TYPE UDT 31
VERSION : 0.0
  STRUCT
   A_FD_OR : BYTE ;	//Feedrate override
   A_DriveEnable : BOOL ;	//Drive test movement enable
   A_AckFixedStop : BOOL ;	//Acknowledge fixed stop reached
   A_SensorFixedStop : BOOL ;	//Sensor fixed stop
   A_ASpDisable : BOOL ;	//Axis/spindle disable
   A_Follow_upMode : BOOL ;	//Follow-up mode
   A_PosMeas1 : BOOL ;	//Position measuring system 1
   A_PosMeas2 : BOOL ;	//Position measuring system 2
   A_ORactive : BOOL ;	//Override active
   A_SWCam : BOOL ;	//SW cam activation
   A_ContrEnable : BOOL ;	//Controller enable
   A_DelDTGSpReset : BOOL ;	//Delete distance to go/Spindle-Reset
   A_Clamp : BOOL ;	//Clamping in progress
   A_RefVal1 : BOOL ;	//Reference point value 1
   A_RefVal2 : BOOL ;	//Reference point value 2
   A_RefVal3 : BOOL ;	//Reference point value 3
   A_RefVal4 : BOOL ;	//Reference point value 4
   A_ExtZO : BOOL ;	//Import external ZO
   A_EnabTravFixedStop : BOOL ;	//Enable travel to fixed stop
   A_FixedFD1 : BOOL ;	//Activate fixed feed 1
   A_FixedFD2 : BOOL ;	//Activate fixed feed 2
   A_FixedFD3 : BOOL ;	//Activate fixed feed 3
   A_FixedFD4 : BOOL ;	//Activate fixed feed 4
   A_VelocSpeedLimit : BOOL ;	//Velocity/spindle speed limitation
   A_PrgtestAxRel : BOOL ;	// Program test axis/spindle release
   A_HW1 : BOOL ;	//Activate handwheel 1
   A_HW2 : BOOL ;	//Activate handwheel 2
   A_HW3 : BOOL ;	//Activate handwheel 3
   A_FDSpStop : BOOL ;	//Feed stop/spindle stop
   A_Disable : BOOL ;	//Traversing key disable
   A_RapidTrOR : BOOL ;	//Rapid traverse override
   A_Minus : BOOL ;	//Traversing key minus
   A_Plus : BOOL ;	//Traversing key plus
   A_INC1 : BOOL ;	//INC1
   A_INC10 : BOOL ;	//INC10
   A_INC100 : BOOL ;	//INC100
   A_INC1000 : BOOL ;	//INC1000
   A_INC10000 : BOOL ;	//INC10000
   A_INCVar : BOOL ;	//INC variable
   A_OEMAxis : BYTE ;	//OEM axis signals
   A_InvHWDirOfRot : BOOL ;	// Inverting handwheel direction of rotation
   f7_1 : BOOL ;
   f7_2 : BOOL ;
   f7_3 : BOOL ;
   f7_4 : BOOL ;
   f7_5 : BOOL ;
   f7_6 : BOOL ;
   f7_7 : BOOL ;
   A_NCASpChanA : BOOL ;	//Assign NC axis/spindle channel A
   A_NCASpChanB : BOOL ;	//Assign NC axis/spindle channel B
   A_NCASpChanC : BOOL ;	//Assign NC axis/spindle channel C
   A_NCASpChanD : BOOL ;	//Assign NC axis/spindle channel D
   A_NCASpStrobe : BOOL ;	//Activation of assignment with pos. edge
   f8_5 : BOOL ;
   f8_6 : BOOL ;
   A_PLCASp : BOOL ;	//Request PLC axis/spindle
   A_Para_A : BOOL ;	//Parameter block servo A
   A_Para_B : BOOL ;	//Parameter block servo B
   A_Para_C : BOOL ;	//Parameter block servo C
   A_LockParSetDef : BOOL ;	//Lock parameter set definition from NC
   f9_4 : BOOL ;
   f9_5 : BOOL ;
   f9_6 : BOOL ;
   f9_7 : BOOL ;
   A_REPOSDelay : BOOL ;	//REPOS DELAY
   f10_1 : BOOL ;
   f10_2 : BOOL ;
   f10_3 : BOOL ;
   f10_4 : BOOL ;
   f10_5 : BOOL ;
   f10_6 : BOOL ;
   f10_7 : BOOL ;
   A_StartBrakeTest : BOOL ;	// Start brake test
   f11_1 : BOOL ;
   f11_2 : BOOL ;
   f11_3 : BOOL ;
   f11_4 : BOOL ;
   f11_5 : BOOL ;
   f11_6 : BOOL ;
   f11_7 : BOOL ;
   A_HWLimitMinus : BOOL ;	//Hardware limit switch minus
   A_HWLimitPlus : BOOL ;	//Hardware limit switch plus
   A_SWLimit2Minus : BOOL ;	//2nd software limit switch minus
   A_SWLimit2Plus : BOOL ;	//2nd software limit switch plus
   A_ModuloLimitEn : BOOL ;	// Modulo limit enabled
   f12_5 : BOOL ;
   f12_6 : BOOL ;
   A_DelayRef : BOOL ;	//Delay reference point approach
   A_JogFixPPos0 : BOOL ;	// JogFixPointPos 0
   A_JogFixPPos1 : BOOL ;	// JogFixPointPos 1
   A_JogFixPPos2 : BOOL ;	// JogFixPointPos 2
   A_JogToPos : BOOL ;	// Jog to position
   f13_4 : BOOL ;
   f13_5 : BOOL ;
   f13_6 : BOOL ;
   f13_7 : BOOL ;
   A_ProgtestSuppress : BOOL ;	// Program test to supress
   A_ProgtestActivate : BOOL ;	// Program test activate
   f14_2 : BOOL ;
   f14_3 : BOOL ;
   f14_4 : BOOL ;
   f14_5 : BOOL ;
   f14_6 : BOOL ;
   f14_7 : BOOL ;
   f15 : BYTE ;
   A_ActGearA : BOOL ;	//Actual gear stage A
   A_ActGearB : BOOL ;	//Actual gear stage B
   A_ActGearC : BOOL ;	//Actual gear stage C
   A_GearChangeOv : BOOL ;	//Gear has changed over
   A_Sp1Syn : BOOL ;	//Re-synchronize spindle 1
   A_Sp2Syn : BOOL ;	//Re-synchronize spindle 2
   A_NoMonitorGear : BOOL ;	//No monitoring when changing gear
   A_DeleteS : BOOL ;	//Delete S value
   A_FD_ORSp : BOOL ;	//Feedrate override for spindle valid
   f17_1 : BOOL ;
   f17_2 : BOOL ;
   f17_3 : BOOL ;
   A_Sp1SynP : BOOL ;	//Re-synchronize spindle 1 f. positioning
   A_Sp2SynP : BOOL ;	//Re-synchronize spindle 2 f. positioning
   A_M3M4Inv : BOOL ;	//Invert M3/M4
   f17_7 : BOOL ;
   f18_0 : BOOL ;
   f18_1 : BOOL ;
   f18_2 : BOOL ;
   f18_3 : BOOL ;
   A_OscilPLC : BOOL ;	//Oscillation via PLC
   A_OscilSpeed : BOOL ;	//enable Oscillation
   A_SetRotDirectRight : BOOL ;	//Setpoint osci. direct. right
   A_SetRotDirectLeft : BOOL ;	//Setpoint osci. direct. left
   A_SpOR : BYTE ;	//Spindle override
   f20_0 : BOOL ;
   A_RUEncQuStop : BOOL ;	//Run-up encoder quick stop
   f20_2 : BOOL ;
   A_SpeedSetpSmooth : BOOL ;	//Speed setpoint smoothing
   f20_4 : BOOL ;
   A_HoldBrakeToOpen : BOOL ;	// holding brake open
   f20_6 : BOOL ;
   f20_7 : BOOL ;
   A_ParA : BOOL ;	//Parameter set selection A
   A_ParB : BOOL ;	//Parameter set selection B
   A_ParC : BOOL ;	//Parameter set selection C
   A_MotA : BOOL ;	//Motor selection A
   A_MotB : BOOL ;	//Motor selection B
   A_MotOK : BOOL ;	//Motor selected
   A_IntegratDisable : BOOL ;	//n controller integrator disable
   A_PulseEnable : BOOL ;	//Pulse enable
   A_SG_SBH : BOOL ;	//Deselection SG/SBH
   A_SBH : BOOL ;	//Deselection of safe standstill
   f22_2 : BOOL ;
   A_SGselect0 : BOOL ;	//Selection SG bit 0
   A_SGselect1 : BOOL ;	//Selection SG bit 1
   f22_5 : BOOL ;
   f22_6 : BOOL ;
   f22_7 : BOOL ;
   A_Transmiss0 : BOOL ;	//Selection Transmission bit 0
   A_Transmiss1 : BOOL ;	//Selection Transmission bit 1
   A_Transmiss2 : BOOL ;	//Selection Transmission bit 2
   f23_3 : BOOL ;
   A_SE : BOOL ;	//Selection SE
   A_BrakeToClose : BOOL ;	//Sinamics: Brake to close
   f23_6 : BOOL ;
   A_TestStop : BOOL ;	//Activate test stop
   A_RotationMonit : BOOL ;	// Stepper motor: Rotation monitoring
   A_ControlAx : BOOL ;	// Control Axis
   f24_2 : BOOL ;
   f24_3 : BOOL ;
   A_TorqComp : BOOL ;	// Torque compensation
   A_ChangSetpOutAss0 : BOOL ;	// Bit value for CTRLOUT_changed - Change setpoint output assignment
   A_ChangSetpOutAss1 : BOOL ;	// Bit value for CTRLOUT_changed - Change setpoint output assignment
   A_MS : BOOL ;	//Master / Slave On
   f25 : BYTE ;
   f26_0 : BOOL ;
   f26_1 : BOOL ;
   f26_2 : BOOL ;
   A_CompContr : BOOL ;	//Compensation controller On
   A_FollowAxOv : BOOL ;	//Enable following axis override
   f26_5 : BOOL ;
   f26_6 : BOOL ;
   f26_7 : BOOL ;
   A_DEPMCS : BOOL ;	// Resume: DEPMCS
   A_DEPBCS : BOOL ;	// Resume: DEPBCS
   A_Corr : BOOL ;	// Resume: Corr
   A_HIAxMove : BOOL ;	// Resume: HIAxMove
   A_StopDEPMCS : BOOL ;	// Stop: DEPMCS
   A_StopDEPBCS : BOOL ;	// Stop: DEPBCS
   A_StopCorr : BOOL ;	// Stop: Corr
   A_StopHIAxMove : BOOL ;	// Stop: HIAxMove
   A_OscillAxExtRev : BOOL ;	// OscillAxExtReversal
   A_AxReset : BOOL ;	// AXRESET
   A_AxResume : BOOL ;	// AXRESUME
   A_SetRP : BOOL ;	//Set reversal point
   A_ChangeRP : BOOL ;	//Change reversal point
   A_StopRP : BOOL ;	//Stop at next reversal point
   A_Stop : BOOL ;	//Stop
   A_PLCAxis : BOOL ;	//PLC checks axis
   f29_0 : BOOL ;
   f29_1 : BOOL ;
   f29_2 : BOOL ;
   f29_3 : BOOL ;
   A_StartGantSynRun : BOOL ;	//Start gantry synchronization run
   A_NoAutoSync : BOOL ;	//No auto sync
   f29_6 : BOOL ;
   f29_7 : BOOL ;
   A_StopSpindle : BOOL ;	//Stop spindle
   A_StartCW : BOOL ;	//Start spindle Clockwise
   A_StartCCW : BOOL ;	//Start spindle Counterclockwise
   A_AutoGearStep : BOOL ;	//Autom. gear step change
   A_PosSpindle : BOOL ;	//Position spindle
   f30_5 : BOOL ;
   f30_6 : BOOL ;
   f30_7 : BOOL ;
   f31_0 : BOOL ;
   f31_1 : BOOL ;
   f31_2 : BOOL ;
   f31_3 : BOOL ;
   A_Resynchronize : BOOL ;	// Resynchronize
   A_DisSync : BOOL ;	// Disable synchronization
   A_Tracksync : BOOL ;	// Track synchronism
   A_DelSyncRunCorr : BOOL ;	// Deleting synchronous run correction
   f32_0 : BOOL ;
   f32_1 : BOOL ;
   A_extStopA : BOOL ;	//Deselection external Stop A
   A_extStopC : BOOL ;	//Deselection external Stop C
   A_extStopD : BOOL ;	//Deselection external Stop D
   A_extStopE : BOOL ;	//Deselection external Stop E
   f32_6 : BOOL ;
   f32_7 : BOOL ;
   f33_0 : BOOL ;
   f33_1 : BOOL ;
   f33_2 : BOOL ;
   f33_3 : BOOL ;
   A_SGcorr_0 : BOOL ;	//Selection SG-correction Bit 0
   A_SGcorr_1 : BOOL ;	//Selection SG-correction Bit 1
   A_SGcorr_2 : BOOL ;	//Selection SG-correction Bit 2
   A_SGcorr_3 : BOOL ;	//Selection SG-correction Bit 3
   f34 : ARRAY  [34 .. 55 ] OF BYTE ;
   A_FeedDriveCAxEng : BOOL ;	// Seperate feed drive as C axis engaged
   A_SpSpeedDisp : BOOL ;	// Spindle speed display
   A_SpInsideClamp : BOOL ;	// Spindle inside clamping
   f56_3 : BOOL ;
   f56_4 : BOOL ;
   f56_5 : BOOL ;
   f56_6 : BOOL ;
   f56_7 : BOOL ;
   f57 : BYTE ;
   f58 : WORD ;	// FC18: internal
   E_SpNA : BOOL ;	//Spindle/no axis
   E_NCU_Link : BOOL ;	//NCU_link active axis
   E_EncodFreq1 : BOOL ;	//Encoder limit frequency 1 exceeded
   E_EncodFreq2 : BOOL ;	//Encoder limit frequency 2 exceeded
   E_RefSyn1 : BOOL ;	//Referenced/synchronized 1
   E_RefSyn2 : BOOL ;	//Referenced/synchronized 2
   E_ExactCoarse : BOOL ;	//Position reached with exact stop coarse
   E_ExactFine : BOOL ;	//Position reached with exact stop fine
   E_TravRequ : BOOL ;	//Travel request
   E_AxialAlarm : BOOL ;	// Axial alarm
   E_AxisReady : BOOL ;	//Axis ready
   E_Follow_upMode : BOOL ;	//Follow-up mode active
   E_Stat : BOOL ;	//Axis/spindle stationary (n<nmin)
   E_PositContr : BOOL ;	//Position controller active
   E_SpeedContr : BOOL ;	//Speed controller active
   E_CurrentContr : BOOL ;	//Current controller active
   E_SWCam : BOOL ;	//Software cams active
   E_HWOverlay : BOOL ;	//Handwheel overlay active
   E_RevFD : BOOL ;	//Revolutional feedrate active
   E_MeasAct : BOOL ;	//Measuring active
   E_ActTravFStop : BOOL ;	//Activate travel to fixed stop
   E_FixedStop : BOOL ;	//Fixed stop reached
   E_ForceFixedStop : BOOL ;	// Force fixed stop limited
   E_AxContainerRot : BOOL ;	// Axis container rotation active
   E_AxReset : BOOL ;	// Axis reset done
   E_PLCCtrlAx : BOOL ;	// PLCcontrolled axis
   E_AxStop : BOOL ;	// Axis stop active
   E_AxSpDisable : BOOL ;	// Axis/spindle disable active
   E_StopDEPMCS : BOOL ;	// stop DEPMCS active
   E_StopDEPBCS : BOOL ;	// stop DEPBCS active
   E_StopCorr : BOOL ;	// stop Corr active
   E_StopHIAxMove : BOOL ;	// Stop HIAxMove active
   E_HW1 : BOOL ;	//Handwheel 1 active
   E_HW2 : BOOL ;	//Handwheel 2 active
   E_HW3 : BOOL ;	//Handwheel 3 active
   f64_3 : BOOL ;
   E_TReqMinus : BOOL ;	// Travel request minus
   E_TReqPlus : BOOL ;	// Travel request plus
   E_TCMinus : BOOL ;	//Traverse command minus
   E_TCPlus : BOOL ;	//Traverse command plus
   E_INC1 : BOOL ;	//INC1
   E_INC10 : BOOL ;	//INC10
   E_INC100 : BOOL ;	//INC100
   E_INC1000 : BOOL ;	//INC1000
   E_INC10000 : BOOL ;	//INC10000
   E_INCVar : BOOL ;	//INC variable
   f65_6 : BOOL ;
   f65_7 : BOOL ;
   E_OEMAxis : BYTE ;	//OEM axis signals
   E_InvHWDirOfRot : BOOL ;	// Handwheel direction of rotation invert actively
   f67_1 : BOOL ;
   f67_2 : BOOL ;
   f67_3 : BOOL ;
   f67_4 : BOOL ;
   f67_5 : BOOL ;
   f67_6 : BOOL ;
   f67_7 : BOOL ;
   E_NCASpChanA : BOOL ;	//NC axis/spindle in channel A
   E_NCASpChanB : BOOL ;	//NC axis/spindle in channel B
   E_NCASpChanC : BOOL ;	//NC axis/spindle in channel C
   E_NCASpChanD : BOOL ;	//NC axis/spindle in channel D
   E_PLCType : BOOL ;	//New type requested by PLC
   E_ChPoss : BOOL ;	//Change axis possible
   E_NeutrASp : BOOL ;	//Neutral axis/spindle
   E_PLCASp : BOOL ;	//PLC axis/spindle
   E_ParS_A : BOOL ;	//Parameter block servo A
   E_ParS_B : BOOL ;	//Parameter block servo B
   E_ParS_C : BOOL ;	//Parameter block servo C
   E_NCUNumLink_3 : BOOL ;
   E_NCUNumLink_4 : BOOL ;
   E_NCUNumLink_5 : BOOL ;
   E_NCUNumLink_6 : BOOL ;
   E_NCUNumLink_7 : BOOL ;
   E_ReposSh : BOOL ;	// Repos shift
   E_ReposShValid : BOOL ;	// Repos shift valid
   E_ReposDelayQuit : BOOL ;	// Repos delay quit
   f70_3 : BOOL ;
   f70_4 : BOOL ;
   f70_5 : BOOL ;
   f70_6 : BOOL ;
   f70_7 : BOOL ;
   E_BrakeTest : BOOL ;	// Brake test active
   f71_1 : BOOL ;
   f71_2 : BOOL ;
   f71_3 : BOOL ;
   E_POS_RESTORED1 : BOOL ;	// POS_RESTORED 1
   E_POS_RESTORED2 : BOOL ;	// POS_RESTORED 2
   f71_6 : BOOL ;
   E_PLCAxDedic : BOOL ;	// PLC Axis dedicated
   E_MMC_REPOSDelay : BOOL ;	//MMC REPOS DELAY
   f72_1 : BOOL ;
   f72_2 : BOOL ;
   f72_3 : BOOL ;
   f72_4 : BOOL ;
   f72_5 : BOOL ;
   f72_6 : BOOL ;
   f72_7 : BOOL ;
   f73 : BYTE ;
   f74_0 : BOOL ;
   f74_1 : BOOL ;
   f74_2 : BOOL ;
   f74_3 : BOOL ;
   E_ModLimEnAct : BOOL ;	// Modulo limit enabled active
   f74_5 : BOOL ;
   f74_6 : BOOL ;
   f74_7 : BOOL ;
   E_JogFixPPos0Act : BOOL ;	// JogFixPointPos 0 active
   E_JogFixPPos1Act : BOOL ;	// JogFixPointPos 1 active
   E_JogFixPPos2Act : BOOL ;	// JogFixPointPos 2 active
   E_JogFixPPos0 : BOOL ;	// JogFixPointPos 0 reached
   E_JogFixPPos1 : BOOL ;	// JogFixPointPos 1 reached
   E_JogFixPPos2 : BOOL ;	// JogFixPointPos 2 reached
   E_JogToPos : BOOL ;	// Jog to position active
   E_JogPos : BOOL ;	// Jog position reached
   E_ScratchPulse : BOOL ;	//Scratch pulse
   f76_1 : BOOL ;
   f76_2 : BOOL ;
   f76_3 : BOOL ;
   E_PathAxis : BOOL ;	// Path axis
   E_PosAxis : BOOL ;	//Positioning axis
   E_IndexAxisPos : BOOL ;	//Indexing axis in position
   E_CurvePos : BOOL ;	//Curve axis in position
   E_CollCheckRedSpeed : BOOL ;	//reduced speed of Collisions Check
   f77_1 : BOOL ;
   f77_2 : BOOL ;
   f77_3 : BOOL ;
   f77_4 : BOOL ;
   f77_5 : BOOL ;
   f77_6 : BOOL ;
   f77_7 : BOOL ;
   E_FPosAxis : REAL ;	//F function (REAL format) for positioning axes
   E_SetpGearA : BOOL ;	//Setpoint gear stage A
   E_SetpGearB : BOOL ;	//Setpoint gear stage B
   E_SetpGearC : BOOL ;	//Setpoint gear stage C
   E_GearChange : BOOL ;	//Gear changeover
   f82_4 : BOOL ;
   f82_5 : BOOL ;
   f82_6 : BOOL ;
   f82_7 : BOOL ;
   E_SpeedLimit : BOOL ;	//Speed limit exceeded
   E_SetSpeedLimit : BOOL ;	//Setpoint speed limited
   E_SetSpeedIncreased : BOOL ;	//Setpoint speed increased
   E_GeoMonit : BOOL ;	//Geometry monitoring
   E_SupportAreaViol : BOOL ;	//Support area limits violated
   E_SetRange : BOOL ;	//Spindle in setpoint range
   E_SpeedMonit : BOOL ;	//Speed monitoring
   E_ActRotRight : BOOL ;	//Actual rotation direction right
   E_ConstCuttSpeed : BOOL ;	//Const. cutting speed active
   E_SUG : BOOL ;	//SUG active (grinding wheel surface speed)
   E_CLG : BOOL ;	//CLG active
   E_Tapping : BOOL ;	//Tapping without compensating chuck
   E_SyncMode : BOOL ;	//Synchronous mode spindle active
   E_PosMode : BOOL ;	//Positioning mode spindle active
   E_OscillMode : BOOL ;	//Oscillation mode spindle active
   E_ContrMode : BOOL ;	//Control mode spindle active
   E_ToolDynLimit : BOOL ;	// Tool with limit of dynamics
   f85_1 : BOOL ;
   f85_2 : BOOL ;
   f85_3 : BOOL ;
   f85_4 : BOOL ;
   E_SpInPosition : BOOL ;	// Spindle in position
   f85_6 : BOOL ;
   f85_7 : BOOL ;
   E_MFunct : INT ;	//M function (INT) for spindle
   E_SFunct : REAL ;	//S function (REAL) for spindle
   f92_0 : BOOL ;
   E_RUEncDisabl : BOOL ;	//Run-up encoder disable active
   f92_2 : BOOL ;
   E_SpeedSetpSmooth : BOOL ;	//Speed setpoint smoothing active
   E_RLIact : BOOL ;	// RLI active
   E_HoldBrakeOpened : BOOL ;	// Holding brake opened
   f92_6 : BOOL ;
   f92_7 : BOOL ;
   E_ParA : BOOL ;	//Active parameter set A
   E_ParB : BOOL ;	//Active parameter set B
   E_ParC : BOOL ;	//Active parameter set C
   E_MotA : BOOL ;	//Active motor A
   E_MotB : BOOL ;	//Active motor B
   E_MotOK : BOOL ;	//Drive ready
   E_IntegratDisable : BOOL ;	//n controller integrator disabled
   E_PulseEnable : BOOL ;	//Pulses enabled
   E_MTempWarn : BOOL ;	//Temperature prewarning motor
   E_HTempWarn : BOOL ;	//Temperature prewarning heat sink
   E_RUComplete : BOOL ;	//Ramp-up complete
   E_MdMdx : BOOL ;	//Md<Mdx
   E_NactNmin : BOOL ;	//nact<nmin
   E_NactNx : BOOL ;	//nact<nx
   E_NactNset : BOOL ;	//nact<nset
   E_Message : BOOL ;	//Variable message function
   E_UDClessAlThreshold : BOOL ;	//UDC-link < alarm threshold
   f95_1 : BOOL ;
   f95_2 : BOOL ;
   f95_3 : BOOL ;
   f95_4 : BOOL ;
   f95_5 : BOOL ;
   f95_6 : BOOL ;
   f95_7 : BOOL ;	// Power Section I2T limit
   E_SpindleMonit : BOOL ;	//Error spindle monitoring
   E_AxisCtrl : BOOL ;	// Axis control active
   E_MSFine : BOOL ;	// Master/Slave fine
   E_MSCoarse : BOOL ;	// Master/Slave coarse
   E_MSCompContr : BOOL ;	// Master/Slave Compensation controller activ
   E_BitValCtrlOutChang0 : BOOL ;	// Bit value for CTRLOUT_changed 0:  Change setpoint output assignment
   E_BitValCtrlOutChang1 : BOOL ;	// Bit value for CTRLOUT_changed 1:  Change setpoint output assignment
   E_MS : BOOL ;	//Master/ slave active
   f97 : BYTE ;
   E_SyncronFine : BOOL ;	//Synchronism fine
   E_SyncronCoarse : BOOL ;	//Synchronism coarse
   E_ActValCoupling : BOOL ;	//Actual value coupling
   f98_3 : BOOL ;
   E_OverlayMotion : BOOL ;	//Overlaid motion
   E_SWL : BOOL ;	//Speed warning limit reached
   E_AWL : BOOL ;	//Acceleration warning limit reached
   E_EmRetr : BOOL ;	//Emergency retraction active
   E_MasterSp : BOOL ;	//Master spindle
   E_SlaveSp : BOOL ;	//Slave spindle
   E_SyncRunCorrDOut : BOOL ;	// Synchronous run correction driven out
   E_AxisAccel : BOOL ;	//Axis accelerated
   E_Sync : BOOL ;	//Synchronization active
   E_MSR : BOOL ;	//Max speed reached
   E_MAR : BOOL ;	//Max acceleration reached
   f99_7 : BOOL ;
   f100_0 : BOOL ;
   f100_1 : BOOL ;
   E_OscillAxExtRev : BOOL ;	// OscillAxExt Reversal active
   E_StopOscill : BOOL ;	//Oscillation cannot start
   E_ErrorOscill : BOOL ;	//Error during oscillation
   E_SparkOut : BOOL ;	//Spark-out active
   E_OscillMotion : BOOL ;	//Oscillation motion active
   E_Oscill : BOOL ;	//Oscillation active
   f101_0 : BOOL ;
   f101_1 : BOOL ;
   E_GantCOLimit : BOOL ;	//Gantry cut-off limit exceeded
   E_GantWarn : BOOL ;	//Gantry warning limit exceeded
   E_SynRunStart : BOOL ;	//Synchronization run ready to start
   E_GantGroupSyn : BOOL ;	//Gantry grouping is synchronous
   E_GantLeadAxis : BOOL ;	//Gantry leading axis
   E_GantAxis : BOOL ;	//Gantry axis
   f102 : BYTE ;
   E_SyncRunCorrIncl : BOOL ;	// Synchronous run correction is included
   f103_1 : BOOL ;
   f103_2 : BOOL ;
   f103_3 : BOOL ;
   f103_4 : BOOL ;
   f103_5 : BOOL ;
   f103_6 : BOOL ;
   f103_7 : BOOL ;
   E_AIAxis : ARRAY  [1 .. 31 ] OF BOOL ;	//Active infeed axis[1..31]
   E_SG_SBH : BOOL ;	//Active SG/SBH
   E_ErrLifeS_CRC : BOOL ;	// Error lifesign or CRC-error
   E_ImpdelNCK : BOOL ;	//Delete pulses NCK
   r108_3 : BOOL ;
   r108_4 : BOOL ;
   r108_5 : BOOL ;
   r108_6 : BOOL ;
   E_SRef : BOOL ;	//Axis safely referenced
   E_SN1Plus : BOOL ;	//Actual position > cam position SN1+
   E_SN1Minus : BOOL ;	//Actual position > cam position SN1-
   E_SN2Plus : BOOL ;	//Actual position > cam position SN2+
   E_SN2Minus : BOOL ;	//Actual position > cam position SN2-
   E_SN3Plus : BOOL ;	//Actual position > cam position SN3+
   E_SN3Minus : BOOL ;	//Actual position > cam position SN3-
   E_SN4Plus : BOOL ;	//Actual position > cam position SN4+
   E_SN4Minus : BOOL ;	//Actual position > cam position SN4-
   f110_0 : BOOL ;
   E_SBH : BOOL ;	//Active SBH
   f110_2 : BOOL ;
   E_SG_0 : BOOL ;	//Active SG 0
   E_SG_1 : BOOL ;	//Active SG 1
   E_n_nx : BOOL ;	//n < nx
   f110_6 : BOOL ;
   f110_7 : BOOL ;
   f111_0 : BOOL ;
   f111_1 : BOOL ;
   f111_2 : BOOL ;
   f111_3 : BOOL ;
   E_StopAB : BOOL ;	//Stop A/B active
   E_StopC : BOOL ;	//Stop C active
   E_StopD : BOOL ;	//Stop D active
   E_StopE : BOOL ;	//Stop E active
   E_CamRangeTr1 : BYTE ;	//Cam Range for Cam Track 1
   E_CamRangeTr2 : BYTE ;	//Cam Range for Cam Track 2
   E_CamRangeTr3 : BYTE ;	//Cam Range for Cam Track 3
   E_CamRangeTr4 : BYTE ;	//Cam Range for Cam Track 4
   f116 : BYTE ;
   E_CamTrack1 : BOOL ;	//Cam Track 1
   E_CamTrack2 : BOOL ;	//Cam Track 2
   E_CamTrack3 : BOOL ;	//Cam Track 3
   E_CamTrack4 : BOOL ;	//Cam Track 4
   f117_4 : BOOL ;
   f117_5 : BOOL ;
   f117_6 : BOOL ;
   f117_7 : BOOL ;
   E_CamRangeBitTr1 : ARRAY  [0 .. 14 ] OF //Cam Range Bits for Cam Track 1
   BOOL ;
   E_CamRangeBitTr2 : ARRAY  [0 .. 14 ] OF //Cam Range Bits for Cam Track 2
   BOOL ;
   E_CamRangeBitTr3 : ARRAY  [0 .. 14 ] OF //Cam Range Bits for Cam Track 3
   BOOL ;
   E_CamRangeBitTr4 : ARRAY  [0 .. 14 ] OF //Cam Range Bits for Cam Track 4
   BOOL ;
   f126 : WORD ;	// internal
   E_MMC_ProgtestSuppress : BOOL ;	// HMI->PLC: Program test to supress
   E_MMC_ProgtestActivate : BOOL ;	// HMI->PLC: Program test activate
   f128_2 : BOOL ;
   f128_3 : BOOL ;
   f128_4 : BOOL ;
   f128_5 : BOOL ;
   f128_6 : BOOL ;
   f128_7 : BOOL ;
   f129 : BYTE ;
   f130 : WORD ;
   E_SensorAv : BOOL ;	// Sensors available
   E_S1aMeasARod : BOOL ;	// Sensor S1: analogous measurement position of actuating rod
   f132_2 : BOOL ;
   f132_3 : BOOL ;
   E_S4dPistonStopP : BOOL ;	// Sensor S4: digital value piston stop position
   E_S5dAngleShaft : BOOL ;	// Sensor S5: digital value angle situation shaft
   f132_6 : BOOL ;
   f132_7 : BOOL ;
   f133 : BYTE ;
   E_ClampingState : INT ;	// state of the clamping system
   E_AnalogSensor : INT ;	// analog sensor on the motor
   f138_0 : BOOL ;
   f138_1 : BOOL ;
   f138_2 : BOOL ;
   f138_3 : BOOL ;
   E_S4PistonStopP : BOOL ;	// Sensor S4: piston stop position
   E_S5AngleShaft : BOOL ;	// Sensor S5: angle situation shaft
   f138_6 : BOOL ;
   f138_7 : BOOL ;
   f139 : BYTE ;
  END_STRUCT ;	
END_TYPE

TYPE UDT 71
VERSION : 0.0
  STRUCT
   IFNo : ARRAY  [1 .. 16 ] OF BOOL ;	//Interface [no.] active
   Quit : ARRAY  [1 .. 16 ] OF BOOL ;	//perform Quit-End
   IF : ARRAY  [1 .. 16 ] OF STRUCT
    Loading : BOOL ;
    Unloading : BOOL ;
    Reloading : BOOL ;
    Positioning : BOOL ;
    PosbyProgram : BOOL ;	//Initiation by CNC Program
    PositioningMT : BOOL ;	//Positioning Multitool
    f0_6 : BOOL ;
    f0_7 : BOOL ;
    PerfStatusError : BOOL ;
    n1_1 : BOOL ;
    n1_2 : BOOL ;
    n1_3 : BOOL ;
    n1_4 : BOOL ;
    n1_5 : BOOL ;
    n1_6 : BOOL ;
    DataInDB1071 : BOOL ;
    Channel : BYTE ;	//Assigned channel
    TMno : BYTE ;	//Tool management no.
    Free1 : DINT ;	//Unassigned parameter 1
    Free2 : DINT ;	//Unassigned parameter 2
    Free3 : DINT ;	//Unassigned parameter 3
    IdentLoad : INT ;	//Identification for loading/unloading station
    NoLoad : INT ;	//No. of loading station
    SMag : INT ;	//Magazine no. (source) for unloading/reloading/pos.
    SLoc : INT ;	//Location no. (source) for unloading/reloading/pos.
    TMag : INT ;	//Magazine no. (target) for loading/reloading
    TLoc : INT ;	//Location no. (target) for loading/reloading
    WithoutMagMoving : BOOL ;	//HMI Data: Without Magazine Moving
    Res2 : BYTE ;
   END_STRUCT ;
  END_STRUCT ;	
END_TYPE

TYPE UDT 72
VERSION : 0.0
  STRUCT
   IFNo : ARRAY  [1 .. 16 ] OF BOOL ;	//Interface [no.] active
   Quit : ARRAY  [1 .. 16 ] OF BOOL ;	//perform Quit-End
   IF : ARRAY  [1 .. 16 ] OF STRUCT
    Comp : BOOL ;	//Compulsory change
    Perform : BOOL ;	//Perform change
    Prepare : BOOL ;	//Prepare change
    T0 : BOOL ;	//T0 programmed
    OldTinDBW42 : BOOL ;	//ZWS No. of Old Tool in DBW (n+42)
    ManTIn : BOOL ;	//Put in Tool in Spindle manual
    ManTOut : BOOL ;	//Get out Tool from Spindle manual
    SpiTRSpi : BOOL ;	//Spindle Tool remains in spindle
    PerfStatusError : BOOL ;
    n1_1 : BOOL ;
    n1_2 : BOOL ;
    n1_3 : BOOL ;
    n1_4 : BOOL ;
    n1_5 : BOOL ;
    n1_6 : BOOL ;
    DataInDB1072 : BOOL ;
    Channel : BYTE ;	//Assigned channel
    TMno : BYTE ;	//Tool management no.
    Free1 : DINT ;	//Unassigned parameter 1
    Free2 : DINT ;	//Unassigned parameter 2
    Free3 : DINT ;	//Unassigned parameter 3
    IdentBuff : INT ;	//Buffer identification (fixed value 9998)
    NoBuff : INT ;	//Relative location (target) in the buffer
    SMag : INT ;	//Magazine no. (source) for new tool
    SLoc : INT ;	//Location no. (source) for new tool
    TMag : INT ;	//Magazine no. (target) for old tool
    TLoc : INT ;	//Location no. (target) for old tool
    LocType : INT ;	//Tool new: location type
    SLeft : INT ;	//Tool new: size left
    SRight : INT ;	//Tool new: size right
    STop : INT ;	//Tool new: size top
    SBottom : INT ;	//Tool new: size bottom
    ToolInBuff : BOOL ;	//ID for tools in buffer
    IgnoreDisab : BOOL ;	//Ignore disabled
    TBUnloaded : BOOL ;	//To be unloaded
    TBLoaded : BOOL ;	//To be loaded
    MasterTool : BOOL ;	//Master tool
    n38_5 : BOOL ;	//reserved
    Exchange_1to1 : BOOL ;	//1:1 exchange
    HandTool : BOOL ;	//Hand tool
    ActTool : BOOL ;	//Active tool
    ToolEnabl : BOOL ;	//Tool enabled
    ToolDisab : BOOL ;	//Tool disabled
    Measured : BOOL ;	//Tool measured
    Prewarn : BOOL ;	//Prewarning limit reached
    ToolChange : BOOL ;	//Tool being changed
    FixedLoc : BOOL ;	//Tool fixed location coded
    ToolUsed : BOOL ;	//Tool was in use
    T_no : INT ;	//Tool new: T no.
    OldTZWSNo : INT ;	//ZWS No. of Old Tool
    MyMag : INT ;
    MyPlace : INT ;
   END_STRUCT ;
  END_STRUCT ;	
END_TYPE

TYPE UDT 73
VERSION : 0.0
  STRUCT
   IfNo : ARRAY  [1 .. 16 ] OF BOOL ;	//Interface [no.] active
   Quit : ARRAY  [1 .. 16 ] OF BOOL ;	//perform Quit-End
   IF : ARRAY  [1 .. 16 ] OF STRUCT
    Comp : BOOL ;	//Compulsory change
    Perform : BOOL ;	//Perform change
    f0_2 : BOOL ;
    T0 : BOOL ;	//T0 programmed
    f0_4 : BOOL ;
    f0_5 : BOOL ;
    ManTOut : BOOL ;	//Get out Tool from Holder manual
    f0_7 : BOOL ;
    PerfStatusError : BOOL ;
    n1_1 : BOOL ;
    n1_2 : BOOL ;
    n1_3 : BOOL ;
    n1_4 : BOOL ;
    n1_5 : BOOL ;
    n1_6 : BOOL ;
    DataInDB1073 : BOOL ;
    Channel : BYTE ;	//Assigned channel
    TMno : BYTE ;	//Tool management no.
    Free1 : DINT ;	//Unassigned parameter 1
    Free2 : DINT ;	//Unassigned parameter 2
    Free3 : DINT ;	//Unassigned parameter 3
    KennZWS : INT ;	//Reserved (buffer identification)
    NoBuff : INT ;	//Rel. location in buffer (res.)
    SMag : INT ;	//Magazine no. of turret
    SLoc : INT ;	//Location no. for new tool
    TMag : INT ;	//Magazine no. of turret (res.)
    TLoc : INT ;	//Location no. for old tool
    LocType : INT ;	//Tool new: location type
    SLeft : INT ;	//Tool new: size left
    SRight : INT ;	//Tool new: size right
    STop : INT ;	//Tool new: size top
    SBottom : INT ;	//Tool new: size bottom
    ToolInBuff : BOOL ;	//ID for tools in buffer
    IgnoreDisab : BOOL ;	//Ignore disabled
    TBUnloaded : BOOL ;	//To be unloaded
    TBLoaded : BOOL ;	//To be loaded
    MasterTool : BOOL ;	//Master tool
    n38_5 : BOOL ;	//reserved
    Exchange_1to1 : BOOL ;	//1:1 exchange
    HandTool : BOOL ;	//Hand tool
    ActTool : BOOL ;	//Active tool
    ToolEnabl : BOOL ;	//Tool enabled
    ToolDisab : BOOL ;	//Tool disabled
    Measured : BOOL ;	//Tool measured
    Prewarn : BOOL ;	//Prewarning limit reached
    ToolChange : BOOL ;	//Tool being changed
    FixedLoc : BOOL ;	//Tool fixed location coded
    ToolUsed : BOOL ;	//Tool was in use
    T_no : INT ;	//Tool new: T no.
    MyPlace : INT ;
   END_STRUCT ;
  END_STRUCT ;	
END_TYPE

TYPE UDT 77
VERSION : 0.0
  STRUCT
   MCP1In : ARRAY  [0 .. 7 ] OF BYTE ;
   MCP1Out : ARRAY  [0 .. 7 ] OF BYTE ;
   MCP1StatSend : DWORD ;
   MCP1StatRec : DWORD ;
   MCP2In : ARRAY  [0 .. 7 ] OF BYTE ;
   MCP2Out : ARRAY  [0 .. 7 ] OF BYTE ;
   MCP2StatSend : DWORD ;
   MCP2StatRec : DWORD ;
   BHGIn : ARRAY  [0 .. 5 ] OF BYTE ;
   Filler : ARRAY  [0 .. 5 ] OF BYTE ;
   BHGOut : ARRAY  [0 .. 19 ] OF BYTE ;
   BHGStatSend : DWORD ;
   BHGStatRec : DWORD ;
  END_STRUCT ;	
END_TYPE

TYPE UDT 1002
VERSION : 0.0
  STRUCT 	//Offset 0
   Chan : ARRAY  [1 .. 10 ] OF STRUCT 	//From Channel 1 to Channel 10
    FDD : ARRAY  [0 .. 15 ] OF //Feed disable
    BOOL ;
    RID : ARRAY  [0 .. 15 ] OF //Read-in disable
    BOOL ;
    NCSD : ARRAY  [0 .. 15 ] OF //NC start disable
    BOOL ;
    FdStop_1 : ARRAY  [0 .. 15 ] OF //Feed stop GEOaxis 1
    BOOL ;
    FdStop_2 : ARRAY  [0 .. 15 ] OF //Feed stop GEOaxis 2
    BOOL ;
    FdStop_3 : ARRAY  [0 .. 15 ] OF //Feed stop GEOaxis 3
    BOOL ;
   END_STRUCT ;	//without Alarmno for Chan (120 Byte)
//Offset 120
   Axis : ARRAY  [1 .. 31 ] OF STRUCT 	//From Axis 1 to Axis 31
    FdStop : ARRAY  [0 .. 15 ] OF //Feed stop axis/spindle 1
    BOOL ;
   END_STRUCT ;	//without Alarmno for Axis (62 Byte)
//Offset 182
   ZInfo0 : ARRAY  [0 .. 63 ] OF WORD ;	//Additional Value for UserAlarms 700000 to 700063
//Offset 310
   ChanA : ARRAY  [1 .. 10 ] OF STRUCT 	//From Channel 1 to Channel 10
    FDD_5C00xx : ARRAY  [0 .. 15 ] OF //Feed disable A.no.51000-510015
    BOOL ;
    FDD_RID_5C01xx : ARRAY  [0 .. 31 ] OF //Feed and read-in disable A.no.510100-510131
    BOOL ;
    RID_5C02xx : ARRAY  [0 .. 31 ] OF //Read-in disable A.no.510200-510231
    BOOL ;
    NCSD_5C03xx : ARRAY  [0 .. 15 ] OF //NC start disable A.no.510300-510315
    BOOL ;
    FdStop_1_5C11xx : ARRAY  [0 .. 15 ] OF //Feed stop GEOaxis 1 A.no.511100-511115
    BOOL ;
    FdStop_2_5C12xx : ARRAY  [0 .. 15 ] OF //Feed stop GEOaxis 2 A.no.511200-511215
    BOOL ;
    FdStop_3_5C13xx : ARRAY  [0 .. 15 ] OF //Feed stop GEOaxis 3 A.no.511300-511315
    BOOL ;
   END_STRUCT ;	//Alarmno for Chan are 5Cxxxx; C is the ChannelNo, except Channel 10. Channel 10
   AxisA : ARRAY  [1 .. 32 ] OF STRUCT 	//From Axis 1 to Axis 31
    AAFdStop60AAxx : ARRAY  [0 .. 15 ] OF //Feed stop axis/spindle
    BOOL ;
   END_STRUCT ;	//Alarmno for Axis are 60AAxx; A is the Axisno.
//Offset 554
   UserA : ARRAY  [0 .. 31 ] OF STRUCT
    A70UUxx : ARRAY  [0 .. 63 ] OF //Alarm 700000-700063 (user area 0)
    BOOL ;
   END_STRUCT ;	//Alarmno for UserAlarms are 7yUUxx; U is the Userarea, y = Db1004.UserDek2No[U]
  END_STRUCT ;	
END_TYPE

TYPE UDT 1071
VERSION : 0.0
  STRUCT
   MTIF : ARRAY  [1 .. 16 ] OF STRUCT
    MtType : INT ;
    MtPlaces : INT ;
    MtDistance : REAL ;
    MtNum : INT ;	// MT-No. to be positioned to
    MtPlaceNum : INT ;	// MT-PlaceNo. ~
    ToolHolder : INT ;	// TH-No as reference for MT-positioning
    IF : ARRAY  [1 .. 3 ] OF STRUCT
     reserved : INT ;	// reserved
    END_STRUCT ;
   END_STRUCT ;
  END_STRUCT ;	
END_TYPE

TYPE UDT 1072
VERSION : 0.0
  STRUCT
   MTIF : ARRAY  [1 .. 16 ] OF STRUCT
    MtType : INT ;
    MtPlaces : INT ;
    MtDistance : REAL ;
    MtNumNew : INT ;	// MT-No. new Tool
    MtPlaceNumNew : INT ;	// MtoolPlaceNum  ~
    MtNumOld : INT ;	// MT-No. old Tool
    MtPlaceNumOld : INT ;	// MtoolPlaceNum  ~
    LocType : INT ;	//Tool new: location type
    SLeft : INT ;	//Tool new: size left
    SRight : INT ;	//Tool new: size right
    STop : INT ;	//Tool new: size top
    SBottom : INT ;	//Tool new: size bottom
    ToolInBuff : BOOL ;	//ID for tools in buffer
    IgnoreDisab : BOOL ;	//Ignore disabled
    TBUnloaded : BOOL ;	//To be unloaded
    TBLoaded : BOOL ;	//To be loaded
    MasterTool : BOOL ;	//Master tool
    n26_5 : BOOL ;	//reserved
    n26_6 : BOOL ;	//reserved
    HandTool : BOOL ;	//Hand tool
    ActTool : BOOL ;	//Active tool
    ToolEnabl : BOOL ;	//Tool enabled
    ToolDisab : BOOL ;	//Tool disabled
    Measured : BOOL ;	//Tool measured
    Prewarn : BOOL ;	//Prewarning limit reached
    ToolChange : BOOL ;	//Tool being changed
    FixedLoc : BOOL ;	//Tool fixed location coded
    ToolUsed : BOOL ;	//Tool was in use
    T_no : INT ;	//Tool new: T no.
    ToolHolder : INT ;	// TH-No as tool compensation reference
    MtMyMag : INT ;	// MtoolNumber the tool is loaded onto
    MtMyPlace : INT ;	// MtoolPlaceNum ~
    IF : ARRAY  [1 .. 7 ] OF STRUCT
     reserved : INT ;	// reserved
    END_STRUCT ;
   END_STRUCT ;
  END_STRUCT ;	
END_TYPE

TYPE UDT 1073
VERSION : 0.0
  STRUCT
   MTIF : ARRAY  [1 .. 16 ] OF STRUCT
    MtType : INT ;
    MtPlaces : INT ;
    MtDistance : REAL ;
    MtNumNew : INT ;	// MT-No. new Tool
    MtPlaceNumNew : INT ;	// MtoolPlaceNum  ~
    MtNumOld : INT ;	// MT-No. old Tool
    MtPlaceNumOld : INT ;	// MtoolPlaceNum  ~
    LocType : INT ;	//Tool new: location type
    SLeft : INT ;	//Tool new: size left
    SRight : INT ;	//Tool new: size right
    STop : INT ;	//Tool new: size top
    SBottom : INT ;	//Tool new: size bottom
    ToolInBuff : BOOL ;	//ID for tools in buffer
    IgnoreDisab : BOOL ;	//Ignore disabled
    TBUnloaded : BOOL ;	//To be unloaded
    TBLoaded : BOOL ;	//To be loaded
    MasterTool : BOOL ;	//Master tool
    n26_5 : BOOL ;	//reserved
    n26_6 : BOOL ;	//reserved
    HandTool : BOOL ;	//Hand tool
    ActTool : BOOL ;	//Active tool
    ToolEnabl : BOOL ;	//Tool enabled
    ToolDisab : BOOL ;	//Tool disabled
    Measured : BOOL ;	//Tool measured
    Prewarn : BOOL ;	//Prewarning limit reached
    ToolChange : BOOL ;	//Tool being changed
    FixedLoc : BOOL ;	//Tool fixed location coded
    ToolUsed : BOOL ;	//Tool was in use
    T_no : INT ;	//Tool new: T no.
    ToolHolder : INT ;	// TH-No as tool compensation reference
    MtMyMag : INT ;	// MtoolNumber the tool is loaded onto
    MtMyPlace : INT ;	// MtoolPlaceNum ~
    IF : ARRAY  [1 .. 7 ] OF STRUCT
     reserved : INT ;	// reserved
    END_STRUCT ;
   END_STRUCT ;
  END_STRUCT ;	
END_TYPE

// FB 1: know-how protected block, not included

// FB 2: know-how protected block, not included

// FB 3: know-how protected block, not included

// FB 4: know-how protected block, not included

// FB 5: know-how protected block, not included

// FB 7: know-how protected block, not included

// FB 9: know-how protected block, not included

// FB 10: know-how protected block, not included

// FB 11: know-how protected block, not included

// FB 29: know-how protected block, not included

// FC 2: know-how protected block, not included

// FC 3: know-how protected block, not included

// FC 5: know-how protected block, not included

// FC 6: know-how protected block, not included

// FC 7: know-how protected block, not included

// FC 8: know-how protected block, not included

// FC 9: know-how protected block, not included

// FC 10: know-how protected block, not included

FUNCTION FC 12 : VOID
AUTHOR : NUMERIK
FAMILY : _800D
NAME : Basics
VERSION : 2.7
VAR_INPUT
  Chan : BYTE ;	//Index of Chan
END_VAR
BEGIN
// (block stored without names or comments; labels and parameter names are numbered)
END_FUNCTION

// FC 13: know-how protected block, not included

// FC 17: know-how protected block, not included

// FC 18: know-how protected block, not included

// FC 19: know-how protected block, not included

// FC 21: know-how protected block, not included

// FC 22: know-how protected block, not included

// FC 24: know-how protected block, not included

// FC 25: know-how protected block, not included

// FC 26: know-how protected block, not included

// FC 1005: know-how protected block, not included

// FC 1006: know-how protected block, not included

DATA_BLOCK DB 4
AUTHOR : NUMERIK
FAMILY : _800D
NAME : Basics
VERSION : 2.7
  STRUCT
   BOfeld0 : WORD  := W#16#CD54;	//Channel 1-8 ever 18 Bits
   BOfeld2 : WORD  := W#16#3553;
   BOfeld4 : WORD  := W#16#D54C;
   BOfeld6 : WORD  := W#16#5533;
   BOfeld8 : WORD  := W#16#55CD;
   BOfeld10 : WORD  := W#16#5435;
   BOfeld12 : WORD  := W#16#53D5;
   BOfeld14 : WORD  := W#16#4C55;
   BOfeld16 : WORD  := W#16#3355;
   BOfeld18 : WORD  := W#16#5555;	//18 Axes/Spindles ever 2 Bit
   BOfeld20 : WORD  := W#16#5555;
   BOfeld22 : WORD  := W#16#F5F0;	//10 User data area ever 8 Bit (Begin: DBB23)
   BOfeld24 : WORD  := W#16#F0F0;
   BOfeld26 : WORD  := W#16#F0F0;
   BOfeld28 : WORD  := W#16#F0F0;
   BOfeld30 : WORD  := W#16#F0F0;
   BOfeld32 : WORD  := W#16#F0F0;
   BOfeld34 : WORD  := W#16#F0F0;
   BOfeld36 : WORD  := W#16#F0F0;
   BOfeld38 : WORD  := W#16#F0F0;
   BOfeld40 : WORD  := W#16#F0F0;
   BOfeld42 : WORD  := W#16#F0F0;
   BOfeld44 : WORD  := W#16#F0F0;
   BOfeld46 : WORD  := W#16#F0F0;
   BOfeld48 : WORD  := W#16#F0F0;
   BOfeld50 : WORD  := W#16#F0F0;
   BOfeld52 : WORD  := W#16#F0F0;
   BOfeld54 : WORD  := W#16#F0F0;
   BOfeld56 : WORD  := W#16#F0F0;
   BOfeld58 : WORD  := W#16#F0F0;
   BOfeld60 : WORD  := W#16#F0F0;
   BOfeld62 : BYTE  := B#16#F0;
   NumUser : BYTE  := B#16#A;
   maganz : BYTE ;	//for TM, number of Magazine
   wzv : BYTE ;
   wzvdat : ARRAY  [1 .. 160 ] OF BYTE ;	//32 Magazine, possibly ever 5 Byte + Spindle
  END_STRUCT ;	
BEGIN
   BOfeld0 := W#16#CD54;
   BOfeld2 := W#16#3553;
   BOfeld4 := W#16#D54C;
   BOfeld6 := W#16#5533;
   BOfeld8 := W#16#55CD;
   BOfeld10 := W#16#5435;
   BOfeld12 := W#16#53D5;
   BOfeld14 := W#16#4C55;
   BOfeld16 := W#16#3355;
   BOfeld18 := W#16#5555;
   BOfeld20 := W#16#5555;
   BOfeld22 := W#16#F5F0;
   BOfeld24 := W#16#F0F0;
   BOfeld26 := W#16#F0F0;
   BOfeld28 := W#16#F0F0;
   BOfeld30 := W#16#F0F0;
   BOfeld32 := W#16#F0F0;
   BOfeld34 := W#16#F0F0;
   BOfeld36 := W#16#F0F0;
   BOfeld38 := W#16#F0F0;
   BOfeld40 := W#16#F0F0;
   BOfeld42 := W#16#F0F0;
   BOfeld44 := W#16#F0F0;
   BOfeld46 := W#16#F0F0;
   BOfeld48 := W#16#F0F0;
   BOfeld50 := W#16#F0F0;
   BOfeld52 := W#16#F0F0;
   BOfeld54 := W#16#F0F0;
   BOfeld56 := W#16#F0F0;
   BOfeld58 := W#16#F0F0;
   BOfeld60 := W#16#F0F0;
   BOfeld62 := B#16#F0;
   NumUser := B#16#A;
END_DATA_BLOCK

DATA_BLOCK DB 5
AUTHOR : NUMERIK
FAMILY : _800D
NAME : Basics
VERSION : 2.7
  STRUCT
   Ch1_DB2_310 : BOOL  := TRUE;	// (Channel 1-10 ever 18 Bits):  error message
   Ch1_DB2_311 : BOOL ;	// Channel 1, DB2.DBB311; operational message
   Ch1_DB2_312 : BOOL  := TRUE;	// Channel 1, DB2.DBB312; error message
   Ch1_DB2_313 : BOOL  := TRUE;	// error message
   Ch1_DB2_314 : BOOL ;	// operational message
   Ch1_DB2_315 : BOOL ;	// operational message
   Ch1_DB2_316 : BOOL  := TRUE;	// error message
   Ch1_DB2_317 : BOOL  := TRUE;	// error message
   Ch1_DB2_318 : BOOL ;	// operational message
   Ch1_DB2_319 : BOOL ;	// operational message
   Ch1_DB2_320 : BOOL  := TRUE;	// error message
   Ch1_DB2_321 : BOOL ;	// operational message
   Ch1_DB2_322 : BOOL  := TRUE;	// error message
   Ch1_DB2_323 : BOOL ;	// operational message
   Ch1_DB2_324 : BOOL  := TRUE;	// error message
   Ch1_DB2_325 : BOOL ;	// operational message
   Ch1_DB2_326 : BOOL  := TRUE;	// error message
   Ch1_DB2_327 : BOOL ;	// operational message
   Ch2_DB2_328 : BOOL  := TRUE;	// Channel 2, DB2.DBB328; error message
   Ch2_DB2_329 : BOOL ;	// Channel 2, DB2.DBB329; operational message
   Ch2_DB2_330 : BOOL  := TRUE;	// error message
   Ch2_DB2_331 : BOOL  := TRUE;	// error message
   Ch2_DB2_332 : BOOL ;	// operational message
   Ch2_DB2_333 : BOOL ;	// operational message
   Ch2_DB2_334 : BOOL  := TRUE;	// error message
   Ch2_DB2_335 : BOOL  := TRUE;	// error message
   Ch2_DB2_336 : BOOL ;	// operational message
   Ch2_DB2_337 : BOOL ;	// operational message
   Ch2_DB2_338 : BOOL  := TRUE;	// error message
   Ch2_DB2_339 : BOOL ;	// operational message
   Ch2_DB2_340 : BOOL  := TRUE;	// error message
   Ch2_DB2_341 : BOOL ;	// operational message
   Ch2_DB2_342 : BOOL  := TRUE;	// error message
   Ch2_DB2_343 : BOOL ;	// operational message
   Ch2_DB2_344 : BOOL  := TRUE;	// error message
   Ch2_DB2_345 : BOOL ;	// operational message
   Ch3_DB2_346 : BOOL  := TRUE;	// Channel 3, DB2.DBB346; error message
   Ch3_DB2_347 : BOOL ;	// Channel 3, DB2.DBB347; operational message
   Ch3_DB2_348 : BOOL  := TRUE;	// error message
   Ch3_DB2_349 : BOOL  := TRUE;	// error message
   Ch3_DB2_350 : BOOL ;	// operational message
   Ch3_DB2_351 : BOOL ;	// operational message
   Ch3_DB2_352 : BOOL  := TRUE;	// error message
   Ch3_DB2_353 : BOOL  := TRUE;	// error message
   Ch3_DB2_354 : BOOL ;	// operational message
   Ch3_DB2_355 : BOOL ;	// operational message
   Ch3_DB2_356 : BOOL  := TRUE;	// error message
   Ch3_DB2_357 : BOOL ;	// operational message
   Ch3_DB2_358 : BOOL  := TRUE;	// error message
   Ch3_DB2_359 : BOOL ;	// operational message
   Ch3_DB2_360 : BOOL  := TRUE;	// error message
   Ch3_DB2_361 : BOOL ;	// operational message
   Ch3_DB2_362 : BOOL  := TRUE;	// error message
   Ch3_DB2_363 : BOOL ;	// operational message
   Ch4_DB2_364 : BOOL  := TRUE;	// Channel 4, DB2.DBB364; error message
   Ch4_DB2_365 : BOOL ;	// Channel 4, DB2.DBB365; operational message
   Ch4_DB2_366 : BOOL  := TRUE;	// error message
   Ch4_DB2_367 : BOOL  := TRUE;	// error message
   Ch4_DB2_368 : BOOL ;	// operational message
   Ch4_DB2_369 : BOOL ;	// operational message
   Ch4_DB2_370 : BOOL  := TRUE;	// error message
   Ch4_DB2_371 : BOOL  := TRUE;	// error message
   Ch4_DB2_372 : BOOL ;	// operational message
   Ch4_DB2_373 : BOOL ;	// operational message
   Ch4_DB2_374 : BOOL  := TRUE;	// error message
   Ch4_DB2_375 : BOOL ;	// operational message
   Ch4_DB2_376 : BOOL  := TRUE;	// error message
   Ch4_DB2_377 : BOOL ;	// operational message
   Ch4_DB2_378 : BOOL  := TRUE;	// error message
   Ch4_DB2_379 : BOOL ;	// operational message
   Ch4_DB2_380 : BOOL  := TRUE;	// error message
   Ch4_DB2_381 : BOOL ;	// operational message
   Ch5_DB2_382 : BOOL  := TRUE;	// Channel 5, DB2.DBB382; error message
   Ch5_DB2_383 : BOOL ;	// Channel 5, DB2.DBB383; operational message
   Ch5_DB2_384 : BOOL  := TRUE;	// error message
   Ch5_DB2_385 : BOOL  := TRUE;	// error message
   Ch5_DB2_386 : BOOL ;	// operational message
   Ch5_DB2_387 : BOOL ;	// operational message
   Ch5_DB2_388 : BOOL  := TRUE;	// error message
   Ch5_DB2_389 : BOOL  := TRUE;	// error message
   Ch5_DB2_390 : BOOL ;	// operational message
   Ch5_DB2_391 : BOOL ;	// operational message
   Ch5_DB2_392 : BOOL  := TRUE;	// error message
   Ch5_DB2_393 : BOOL ;	// operational message
   Ch5_DB2_394 : BOOL  := TRUE;	// error message
   Ch5_DB2_395 : BOOL ;	// operational message
   Ch5_DB2_396 : BOOL  := TRUE;	// error message
   Ch5_DB2_397 : BOOL ;	// operational message
   Ch5_DB2_398 : BOOL  := TRUE;	// error message
   Ch5_DB2_399 : BOOL ;	// operational message
   Ch6_DB2_400 : BOOL  := TRUE;	// Channel 6, DB2.DBB400; error message
   Ch6_DB2_401 : BOOL ;	// Channel 6, DB2.DBB401; operational message
   Ch6_DB2_402 : BOOL  := TRUE;	// error message
   Ch6_DB2_403 : BOOL  := TRUE;	// error message
   Ch6_DB2_404 : BOOL ;	// operational message
   Ch6_DB2_405 : BOOL ;	// operational message
   Ch6_DB2_406 : BOOL  := TRUE;	// error message
   Ch6_DB2_407 : BOOL  := TRUE;	// error message
   Ch6_DB2_408 : BOOL ;	// operational message
   Ch6_DB2_409 : BOOL ;	// operational message
   Ch6_DB2_410 : BOOL  := TRUE;	// error message
   Ch6_DB2_411 : BOOL ;	// operational message
   Ch6_DB2_412 : BOOL  := TRUE;	// error message
   Ch6_DB2_413 : BOOL ;	// operational message
   Ch6_DB2_414 : BOOL  := TRUE;	// error message
   Ch6_DB2_415 : BOOL ;	// operational message
   Ch6_DB2_416 : BOOL  := TRUE;	// error message
   Ch6_DB2_417 : BOOL ;	// operational message
   Ch7_DB2_418 : BOOL  := TRUE;	// Channel 7, DB2.DBB418; error message
   Ch7_DB2_419 : BOOL ;	// Channel 7, DB2.DBB419; operational message
   Ch7_DB2_420 : BOOL  := TRUE;	// error message
   Ch7_DB2_421 : BOOL  := TRUE;	// error message
   Ch7_DB2_422 : BOOL ;	// operational message
   Ch7_DB2_423 : BOOL ;	// operational message
   Ch7_DB2_424 : BOOL  := TRUE;	// error message
   Ch7_DB2_425 : BOOL  := TRUE;	// error message
   Ch7_DB2_426 : BOOL ;	// operational message
   Ch7_DB2_427 : BOOL ;	// operational message
   Ch7_DB2_428 : BOOL  := TRUE;	// error message
   Ch7_DB2_429 : BOOL ;	// operational message
   Ch7_DB2_430 : BOOL  := TRUE;	// error message
   Ch7_DB2_431 : BOOL ;	// operational message
   Ch7_DB2_432 : BOOL  := TRUE;	// error message
   Ch7_DB2_433 : BOOL ;	// operational message
   Ch7_DB2_434 : BOOL  := TRUE;	// error message
   Ch7_DB2_435 : BOOL ;	// operational message
   Ch8_DB2_436 : BOOL  := TRUE;	// Channel 8, DB2.DBB436; error message
   Ch8_DB2_437 : BOOL ;	// Channel 8, DB2.DBB437; operational message
   Ch8_DB2_438 : BOOL  := TRUE;	// error message
   Ch8_DB2_439 : BOOL  := TRUE;	// error message
   Ch8_DB2_440 : BOOL ;	// operational message
   Ch8_DB2_441 : BOOL ;	// operational message
   Ch8_DB2_442 : BOOL  := TRUE;	// error message
   Ch8_DB2_443 : BOOL  := TRUE;	// error message
   Ch8_DB2_444 : BOOL ;	// operational message
   Ch8_DB2_445 : BOOL ;	// operational message
   Ch8_DB2_446 : BOOL  := TRUE;	// error message
   Ch8_DB2_447 : BOOL ;	// operational message
   Ch8_DB2_448 : BOOL  := TRUE;	// error message
   Ch8_DB2_449 : BOOL ;	// operational message
   Ch8_DB2_450 : BOOL  := TRUE;	// error message
   Ch8_DB2_451 : BOOL ;	// operational message
   Ch8_DB2_452 : BOOL  := TRUE;	// error message
   Ch8_DB2_453 : BOOL ;	// operational message
   Ch9_DB2_454 : BOOL  := TRUE;	// Channel 9, DB2.DBB454; error message
   Ch9_DB2_455 : BOOL ;	// Channel 9, DB2.DBB455; operational message
   Ch9_DB2_456 : BOOL  := TRUE;	// error message
   Ch9_DB2_457 : BOOL  := TRUE;	// error message
   Ch9_DB2_458 : BOOL ;	// operational message
   Ch9_DB2_459 : BOOL ;	// operational message
   Ch9_DB2_460 : BOOL  := TRUE;	// error message
   Ch9_DB2_461 : BOOL  := TRUE;	// error message
   Ch9_DB2_462 : BOOL ;	// operational message
   Ch9_DB2_463 : BOOL ;	// operational message
   Ch9_DB2_464 : BOOL  := TRUE;	// error message
   Ch9_DB2_465 : BOOL ;	// operational message
   Ch9_DB2_466 : BOOL  := TRUE;	// error message
   Ch9_DB2_467 : BOOL ;	// operational message
   Ch9_DB2_468 : BOOL  := TRUE;	// error message
   Ch9_DB2_469 : BOOL ;	// operational message
   Ch9_DB2_470 : BOOL  := TRUE;	// error message
   Ch9_DB2_471 : BOOL ;	// operational message
   Ch10_DB2_472 : BOOL  := TRUE;	// Channel 10, DB2.DBB472; error message
   Ch10_DB2_473 : BOOL ;	// Channel 10, DB2.DBB473; operational message
   Ch10_DB2_474 : BOOL  := TRUE;	// error message
   Ch10_DB2_475 : BOOL  := TRUE;	// error message
   Ch10_DB2_476 : BOOL ;	// operational message
   Ch10_DB2_477 : BOOL ;	// operational message
   Ch10_DB2_478 : BOOL  := TRUE;	// error message
   Ch10_DB2_479 : BOOL  := TRUE;	// error message
   Ch10_DB2_480 : BOOL ;	// operational message
   Ch10_DB2_481 : BOOL ;	// operational message
   Ch10_DB2_482 : BOOL  := TRUE;	// error message
   Ch10_DB2_483 : BOOL ;	// operational message
   Ch10_DB2_484 : BOOL  := TRUE;	// error message
   Ch10_DB2_485 : BOOL ;	// operational message
   Ch10_DB2_486 : BOOL  := TRUE;	// error message
   Ch10_DB2_487 : BOOL ;	// operational message
   Ch10_DB2_488 : BOOL  := TRUE;	// error message
   Ch10_DB2_489 : BOOL ;	// operational message
   Ax1_DB2_490 : BOOL  := TRUE;	// (32 Axes/Spindles ever 2 Bit):  error message
   Ax1_DB2_491 : BOOL ;	// Axis 1, DB2.DBB491; operational message
   Ax2_DB2_492 : BOOL  := TRUE;	// Axis 2, DB2.DBB492; error message
   Ax2_DB2_493 : BOOL ;	// Axis 2, DB2.DBB493; operational message
   Ax3_DB2_494 : BOOL  := TRUE;	// error message
   Ax3_DB2_495 : BOOL ;	// operational message
   Ax4_DB2_496 : BOOL  := TRUE;	// error message
   Ax4_DB2_497 : BOOL ;	// operational message
   Ax5_DB2_498 : BOOL  := TRUE;	// error message
   Ax5_DB2_499 : BOOL ;	// operational message
   Ax6_DB2_500 : BOOL  := TRUE;	// error message
   Ax6_DB2_501 : BOOL ;	// operational message
   Ax7_DB2_502 : BOOL  := TRUE;	// error message
   Ax7_DB2_503 : BOOL ;	// operational message
   Ax8_DB2_504 : BOOL  := TRUE;	// error message
   Ax8_DB2_505 : BOOL ;	// operational message
   Ax9_DB2_506 : BOOL  := TRUE;	// error message
   Ax9_DB2_507 : BOOL ;	// operational message
   Ax10_DB2_508 : BOOL  := TRUE;	// error message
   Ax10_DB2_509 : BOOL ;	// operational message
   Ax11_DB2_510 : BOOL  := TRUE;	// error message
   Ax11_DB2_511 : BOOL ;	// operational message
   Ax12_DB2_512 : BOOL  := TRUE;	// error message
   Ax12_DB2_513 : BOOL ;	// operational message
   Ax13_DB2_514 : BOOL  := TRUE;	// error message
   Ax13_DB2_515 : BOOL ;	// operational message
   Ax14_DB2_516 : BOOL  := TRUE;	// error message
   Ax14_DB2_517 : BOOL ;	// operational message
   Ax15_DB2_518 : BOOL  := TRUE;	// error message
   Ax15_DB2_519 : BOOL ;	// operational message
   Ax16_DB2_520 : BOOL  := TRUE;	// error message
   Ax16_DB2_521 : BOOL ;	// operational message
   Ax17_DB2_522 : BOOL  := TRUE;	// error message
   Ax17_DB2_523 : BOOL ;	// operational message
   Ax18_DB2_524 : BOOL  := TRUE;	// error message
   Ax18_DB2_525 : BOOL ;	// operational message
   Ax19_DB2_526 : BOOL  := TRUE;	// error message
   Ax19_DB2_527 : BOOL ;	// operational message
   Ax20_DB2_528 : BOOL  := TRUE;	// error message
   Ax20_DB2_529 : BOOL ;	// operational message
   Ax21_DB2_530 : BOOL  := TRUE;	// error message
   Ax21_DB2_531 : BOOL ;	// operational message
   Ax22_DB2_532 : BOOL  := TRUE;	// error message
   Ax22_DB2_533 : BOOL ;	// operational message
   Ax23_DB2_534 : BOOL  := TRUE;	// error message
   Ax23_DB2_535 : BOOL ;	// operational message
   Ax24_DB2_536 : BOOL  := TRUE;	// error message
   Ax24_DB2_537 : BOOL ;	// operational message
   Ax25_DB2_538 : BOOL  := TRUE;	// error message
   Ax25_DB2_539 : BOOL ;	// operational message
   Ax26_DB2_540 : BOOL  := TRUE;	// error message
   Ax26_DB2_541 : BOOL ;	// operational message
   Ax27_DB2_542 : BOOL  := TRUE;	// error message
   Ax27_DB2_543 : BOOL ;	// operational message
   Ax28_DB2_544 : BOOL  := TRUE;	// error message
   Ax28_DB2_545 : BOOL ;	// operational message
   Ax29_DB2_546 : BOOL  := TRUE;	// error message
   Ax29_DB2_547 : BOOL ;	// operational message
   Ax30_DB2_548 : BOOL  := TRUE;	// error message
   Ax30_DB2_549 : BOOL ;	// operational message
   Ax31_DB2_550 : BOOL  := TRUE;	// error message
   Ax31_DB2_551 : BOOL ;	// operational message
   Ax32_DB2_552 : BOOL  := TRUE;	// error message
   Ax32_DB2_553 : BOOL ;	// operational message
   User0_DB2_554 : BOOL  := TRUE;	// (32 User data area ever 8 Bit):  error message
   User0_DB2_555 : BOOL  := TRUE;	// UserDataArea 0, DB2.DBB555; error message
   User0_DB2_556 : BOOL  := TRUE;	// error message
   User0_DB2_557 : BOOL  := TRUE;	// error message
   User0_DB2_558 : BOOL ;	// operational message
   User0_DB2_559 : BOOL ;	// operational message
   User0_DB2_560 : BOOL ;	// operational message
   User0_DB2_561 : BOOL ;	// operational message
   User1_DB2_562 : BOOL  := TRUE;	// UserDataArea 1, DB2.DBB562; error message
   User1_DB2_563 : BOOL  := TRUE;	// error message
   User1_DB2_564 : BOOL  := TRUE;	// error message
   User1_DB2_565 : BOOL  := TRUE;	// error message
   User1_DB2_566 : BOOL ;	// operational message
   User1_DB2_567 : BOOL ;	// operational message
   User1_DB2_568 : BOOL ;	// operational message
   User1_DB2_569 : BOOL ;	// operational message
   User2_DB2_570 : BOOL  := TRUE;	// UserDataArea 2, DB2.DBB570; error message
   User2_DB2_571 : BOOL  := TRUE;	// error message
   User2_DB2_572 : BOOL  := TRUE;	// error message
   User2_DB2_573 : BOOL  := TRUE;	// error message
   User2_DB2_574 : BOOL ;	// operational message
   User2_DB2_575 : BOOL ;	// operational message
   User2_DB2_576 : BOOL ;	// operational message
   User2_DB2_577 : BOOL ;	// operational message
   User3_DB2_578 : BOOL  := TRUE;	// UserDataArea 3, DB2.DBB578; error message
   User3_DB2_579 : BOOL  := TRUE;	// error message
   User3_DB2_580 : BOOL  := TRUE;	// error message
   User3_DB2_581 : BOOL  := TRUE;	// error message
   User3_DB2_582 : BOOL ;	// operational message
   User3_DB2_583 : BOOL ;	// operational message
   User3_DB2_584 : BOOL ;	// operational message
   User3_DB2_585 : BOOL ;	// operational message
   User4_DB2_586 : BOOL  := TRUE;	// UserDataArea 4, DB2.DBB586; error message
   User4_DB2_587 : BOOL  := TRUE;	// error message
   User4_DB2_588 : BOOL  := TRUE;	// error message
   User4_DB2_589 : BOOL  := TRUE;	// error message
   User4_DB2_590 : BOOL ;	// operational message
   User4_DB2_591 : BOOL ;	// operational message
   User4_DB2_592 : BOOL ;	// operational message
   User4_DB2_593 : BOOL ;	// operational message
   User5_DB2_594 : BOOL  := TRUE;	// UserDataArea 5, DB2.DBB594; error message
   User5_DB2_595 : BOOL  := TRUE;	// error message
   User5_DB2_596 : BOOL  := TRUE;	// error message
   User5_DB2_597 : BOOL  := TRUE;	// error message
   User5_DB2_598 : BOOL ;	// operational message
   User5_DB2_599 : BOOL ;	// operational message
   User5_DB2_600 : BOOL ;	// operational message
   User5_DB2_601 : BOOL ;	// operational message
   User6_DB2_602 : BOOL  := TRUE;	// UserDataArea 6, DB2.DBB602; error message
   User6_DB2_603 : BOOL  := TRUE;	// error message
   User6_DB2_604 : BOOL  := TRUE;	// error message
   User6_DB2_605 : BOOL  := TRUE;	// error message
   User6_DB2_606 : BOOL ;	// operational message
   User6_DB2_607 : BOOL ;	// operational message
   User6_DB2_608 : BOOL ;	// operational message
   User6_DB2_609 : BOOL ;	// operational message
   User7_DB2_610 : BOOL  := TRUE;	// UserDataArea 7, DB2.DBB610; error message
   User7_DB2_611 : BOOL  := TRUE;	// error message
   User7_DB2_612 : BOOL  := TRUE;	// error message
   User7_DB2_613 : BOOL  := TRUE;	// error message
   User7_DB2_614 : BOOL ;	// operational message
   User7_DB2_615 : BOOL ;	// operational message
   User7_DB2_616 : BOOL ;	// operational message
   User7_DB2_617 : BOOL ;	// operational message
   User8_DB2_618 : BOOL  := TRUE;	// UserDataArea 8, DB2.DBB618; error message
   User8_DB2_619 : BOOL  := TRUE;	// error message
   User8_DB2_620 : BOOL  := TRUE;	// error message
   User8_DB2_621 : BOOL  := TRUE;	// error message
   User8_DB2_622 : BOOL ;	// operational message
   User8_DB2_623 : BOOL ;	// operational message
   User8_DB2_624 : BOOL ;	// operational message
   User8_DB2_625 : BOOL ;	// operational message
   User9_DB2_626 : BOOL  := TRUE;	// UserDataArea 9, DB2.DBB626; error message
   User9_DB2_627 : BOOL  := TRUE;	// error message
   User9_DB2_628 : BOOL  := TRUE;	// error message
   User9_DB2_629 : BOOL  := TRUE;	// error message
   User9_DB2_630 : BOOL ;	// operational message
   User9_DB2_631 : BOOL ;	// operational message
   User9_DB2_632 : BOOL ;	// operational message
   User9_DB2_633 : BOOL ;	// operational message
   User10_DB2_634 : BOOL  := TRUE;	// UserDataArea 10, DB2.DBB634; error message
   User10_DB2_635 : BOOL  := TRUE;	// error message
   User10_DB2_636 : BOOL  := TRUE;	// error message
   User10_DB2_637 : BOOL  := TRUE;	// error message
   User10_DB2_638 : BOOL ;	// operational message
   User10_DB2_639 : BOOL ;	// operational message
   User10_DB2_640 : BOOL ;	// operational message
   User10_DB2_641 : BOOL ;	// operational message
   User11_DB2_642 : BOOL  := TRUE;	// UserDataArea 11, DB2.DBB642; error message
   User11_DB2_643 : BOOL  := TRUE;	// error message
   User11_DB2_644 : BOOL  := TRUE;	// error message
   User11_DB2_645 : BOOL  := TRUE;	// error message
   User11_DB2_646 : BOOL ;	// operational message
   User11_DB2_647 : BOOL ;	// operational message
   User11_DB2_648 : BOOL ;	// operational message
   User11_DB2_649 : BOOL ;	// operational message
   User12_DB2_650 : BOOL  := TRUE;	// UserDataArea 12, DB2.DBB650; error message
   User12_DB2_651 : BOOL  := TRUE;	// error message
   User12_DB2_652 : BOOL  := TRUE;	// error message
   User12_DB2_653 : BOOL  := TRUE;	// error message
   User12_DB2_654 : BOOL ;	// operational message
   User12_DB2_655 : BOOL ;	// operational message
   User12_DB2_656 : BOOL ;	// operational message
   User12_DB2_657 : BOOL ;	// operational message
   User13_DB2_658 : BOOL  := TRUE;	// UserDataArea 13, DB2.DBB658; error message
   User13_DB2_659 : BOOL  := TRUE;	// error message
   User13_DB2_660 : BOOL  := TRUE;	// error message
   User13_DB2_661 : BOOL  := TRUE;	// error message
   User13_DB2_662 : BOOL ;	// operational message
   User13_DB2_663 : BOOL ;	// operational message
   User13_DB2_664 : BOOL ;	// operational message
   User13_DB2_665 : BOOL ;	// operational message
   User14_DB2_666 : BOOL  := TRUE;	// UserDataArea 14, DB2.DBB666; error message
   User14_DB2_667 : BOOL  := TRUE;	// error message
   User14_DB2_668 : BOOL  := TRUE;	// error message
   User14_DB2_669 : BOOL  := TRUE;	// error message
   User14_DB2_670 : BOOL ;	// operational message
   User14_DB2_671 : BOOL ;	// operational message
   User14_DB2_672 : BOOL ;	// operational message
   User14_DB2_673 : BOOL ;	// operational message
   User15_DB2_674 : BOOL  := TRUE;	// UserDataArea 15, DB2.DBB674; error message
   User15_DB2_675 : BOOL  := TRUE;	// error message
   User15_DB2_676 : BOOL  := TRUE;	// error message
   User15_DB2_677 : BOOL  := TRUE;	// error message
   User15_DB2_678 : BOOL ;	// operational message
   User15_DB2_679 : BOOL ;	// operational message
   User15_DB2_680 : BOOL ;	// operational message
   User15_DB2_681 : BOOL ;	// operational message
   User16_DB2_682 : BOOL  := TRUE;	// UserDataArea 16, DB2.DBB682; error message
   User16_DB2_683 : BOOL  := TRUE;	// error message
   User16_DB2_684 : BOOL  := TRUE;	// error message
   User16_DB2_685 : BOOL  := TRUE;	// error message
   User16_DB2_686 : BOOL ;	// operational message
   User16_DB2_687 : BOOL ;	// operational message
   User16_DB2_688 : BOOL ;	// operational message
   User16_DB2_689 : BOOL ;	// operational message
   User17_DB2_690 : BOOL  := TRUE;	// UserDataArea 17, DB2.DBB690; error message
   User17_DB2_691 : BOOL  := TRUE;	// error message
   User17_DB2_692 : BOOL  := TRUE;	// error message
   User17_DB2_693 : BOOL  := TRUE;	// error message
   User17_DB2_694 : BOOL ;	// operational message
   User17_DB2_695 : BOOL ;	// operational message
   User17_DB2_696 : BOOL ;	// operational message
   User17_DB2_697 : BOOL ;	// operational message
   User18_DB2_698 : BOOL  := TRUE;	// UserDataArea 18, DB2.DBB698; error message
   User18_DB2_699 : BOOL  := TRUE;	// error message
   User18_DB2_700 : BOOL  := TRUE;	// error message
   User18_DB2_701 : BOOL  := TRUE;	// error message
   User18_DB2_702 : BOOL ;	// operational message
   User18_DB2_703 : BOOL ;	// operational message
   User18_DB2_704 : BOOL ;	// operational message
   User18_DB2_705 : BOOL ;	// operational message
   User19_DB2_706 : BOOL  := TRUE;	// UserDataArea 19, DB2.DBB706; error message
   User19_DB2_707 : BOOL  := TRUE;	// error message
   User19_DB2_708 : BOOL  := TRUE;	// error message
   User19_DB2_709 : BOOL  := TRUE;	// error message
   User19_DB2_710 : BOOL ;	// operational message
   User19_DB2_711 : BOOL ;	// operational message
   User19_DB2_712 : BOOL ;	// operational message
   User19_DB2_713 : BOOL ;	// operational message
   User20_DB2_714 : BOOL  := TRUE;	// UserDataArea 20, DB2.DBB714; error message
   User20_DB2_715 : BOOL  := TRUE;	// error message
   User20_DB2_716 : BOOL  := TRUE;	// error message
   User20_DB2_717 : BOOL  := TRUE;	// error message
   User20_DB2_718 : BOOL ;	// operational message
   User20_DB2_719 : BOOL ;	// operational message
   User20_DB2_720 : BOOL ;	// operational message
   User20_DB2_721 : BOOL ;	// operational message
   User21_DB2_722 : BOOL  := TRUE;	// UserDataArea 21, DB2.DBB722; error message
   User21_DB2_723 : BOOL  := TRUE;	// error message
   User21_DB2_724 : BOOL  := TRUE;	// error message
   User21_DB2_725 : BOOL  := TRUE;	// error message
   User21_DB2_726 : BOOL ;	// operational message
   User21_DB2_727 : BOOL ;	// operational message
   User21_DB2_728 : BOOL ;	// operational message
   User21_DB2_729 : BOOL ;	// operational message
   User22_DB2_730 : BOOL  := TRUE;	// UserDataArea 22, DB2.DBB730; error message
   User22_DB2_731 : BOOL  := TRUE;	// error message
   User22_DB2_732 : BOOL  := TRUE;	// error message
   User22_DB2_733 : BOOL  := TRUE;	// error message
   User22_DB2_734 : BOOL ;	// operational message
   User22_DB2_735 : BOOL ;	// operational message
   User22_DB2_736 : BOOL ;	// operational message
   User22_DB2_737 : BOOL ;	// operational message
   User23_DB2_738 : BOOL  := TRUE;	// UserDataArea 23, DB2.DBB738; error message
   User23_DB2_739 : BOOL  := TRUE;	// error message
   User23_DB2_740 : BOOL  := TRUE;	// error message
   User23_DB2_741 : BOOL  := TRUE;	// error message
   User23_DB2_742 : BOOL ;	// operational message
   User23_DB2_743 : BOOL ;	// operational message
   User23_DB2_744 : BOOL ;	// operational message
   User23_DB2_745 : BOOL ;	// operational message
   User24_DB2_746 : BOOL  := TRUE;	// UserDataArea 24, DB2.DBB746; error message
   User24_DB2_747 : BOOL  := TRUE;	// error message
   User24_DB2_748 : BOOL  := TRUE;	// error message
   User24_DB2_749 : BOOL  := TRUE;	// error message
   User24_DB2_750 : BOOL ;	// operational message
   User24_DB2_751 : BOOL ;	// operational message
   User24_DB2_752 : BOOL ;	// operational message
   User24_DB2_753 : BOOL ;	// operational message
   User25_DB2_754 : BOOL  := TRUE;	// UserDataArea 25, DB2.DBB754; error message
   User25_DB2_755 : BOOL  := TRUE;	// error message
   User25_DB2_756 : BOOL  := TRUE;	// error message
   User25_DB2_757 : BOOL  := TRUE;	// error message
   User25_DB2_758 : BOOL ;	// operational message
   User25_DB2_759 : BOOL ;	// operational message
   User25_DB2_760 : BOOL ;	// operational message
   User25_DB2_761 : BOOL ;	// operational message
   User26_DB2_762 : BOOL  := TRUE;	// UserDataArea 26, DB2.DBB762; error message
   User26_DB2_763 : BOOL  := TRUE;	// error message
   User26_DB2_764 : BOOL  := TRUE;	// error message
   User26_DB2_765 : BOOL  := TRUE;	// error message
   User26_DB2_766 : BOOL ;	// operational message
   User26_DB2_767 : BOOL ;	// operational message
   User26_DB2_768 : BOOL ;	// operational message
   User26_DB2_769 : BOOL ;	// operational message
   User27_DB2_770 : BOOL  := TRUE;	// UserDataArea 27, DB2.DBB770; error message
   User27_DB2_771 : BOOL  := TRUE;	// error message
   User27_DB2_772 : BOOL  := TRUE;	// error message
   User27_DB2_773 : BOOL  := TRUE;	// error message
   User27_DB2_774 : BOOL ;	// operational message
   User27_DB2_775 : BOOL ;	// operational message
   User27_DB2_776 : BOOL ;	// operational message
   User27_DB2_777 : BOOL ;	// operational message
   User28_DB2_778 : BOOL  := TRUE;	// UserDataArea 28, DB2.DBB778; error message
   User28_DB2_779 : BOOL  := TRUE;	// error message
   User28_DB2_780 : BOOL  := TRUE;	// error message
   User28_DB2_781 : BOOL  := TRUE;	// error message
   User28_DB2_782 : BOOL ;	// operational message
   User28_DB2_783 : BOOL ;	// operational message
   User28_DB2_784 : BOOL ;	// operational message
   User28_DB2_785 : BOOL ;	// operational message
   User29_DB2_786 : BOOL  := TRUE;	// UserDataArea 29, DB2.DBB786; error message
   User29_DB2_787 : BOOL  := TRUE;	// error message
   User29_DB2_788 : BOOL  := TRUE;	// error message
   User29_DB2_789 : BOOL  := TRUE;	// error message
   User29_DB2_790 : BOOL ;	// operational message
   User29_DB2_791 : BOOL ;	// operational message
   User29_DB2_792 : BOOL ;	// operational message
   User29_DB2_793 : BOOL ;	// operational message
   User30_DB2_794 : BOOL  := TRUE;	// UserDataArea 30, DB2.DBB794; error message
   User30_DB2_795 : BOOL  := TRUE;	// error message
   User30_DB2_796 : BOOL  := TRUE;	// error message
   User30_DB2_797 : BOOL  := TRUE;	// error message
   User30_DB2_798 : BOOL ;	// operational message
   User30_DB2_799 : BOOL ;	// operational message
   User30_DB2_800 : BOOL ;	// operational message
   User30_DB2_801 : BOOL ;	// operational message
   User31_DB2_802 : BOOL  := TRUE;	// UserDataArea 31, DB2.DBB802; error message
   User31_DB2_803 : BOOL  := TRUE;	// error message
   User31_DB2_804 : BOOL  := TRUE;	// error message
   User31_DB2_805 : BOOL  := TRUE;	// error message
   User31_DB2_806 : BOOL ;	// operational message
   User31_DB2_807 : BOOL ;	// operational message
   User31_DB2_808 : BOOL ;	// operational message
   User31_DB2_809 : BOOL ;	// operational message
   Bit62_4 : BOOL ;	// reserved
   Bit62_5 : BOOL ;	// reserved
   Bit62_6 : BOOL ;	// reserved
   Bit62_7 : BOOL ;	// reserved
   Byte63 : BYTE ;	// reserved
   Word64 : WORD ;	// reserved
   Word66 : WORD ;	// reserved
   Word68 : WORD ;	// reserved
   Word70 : WORD ;	// reserved
   UserDek2No : ARRAY  [0 .. 31 ] OF // UserDek2No: Value 0..9 possible
   BYTE  := B#16#0;
  END_STRUCT ;	
BEGIN
   Ch1_DB2_310 := TRUE;
   Ch1_DB2_312 := TRUE;
   Ch1_DB2_313 := TRUE;
   Ch1_DB2_316 := TRUE;
   Ch1_DB2_317 := TRUE;
   Ch1_DB2_320 := TRUE;
   Ch1_DB2_322 := TRUE;
   Ch1_DB2_324 := TRUE;
   Ch1_DB2_326 := TRUE;
   Ch2_DB2_328 := TRUE;
   Ch2_DB2_330 := TRUE;
   Ch2_DB2_331 := TRUE;
   Ch2_DB2_334 := TRUE;
   Ch2_DB2_335 := TRUE;
   Ch2_DB2_338 := TRUE;
   Ch2_DB2_340 := TRUE;
   Ch2_DB2_342 := TRUE;
   Ch2_DB2_344 := TRUE;
   Ch3_DB2_346 := TRUE;
   Ch3_DB2_348 := TRUE;
   Ch3_DB2_349 := TRUE;
   Ch3_DB2_352 := TRUE;
   Ch3_DB2_353 := TRUE;
   Ch3_DB2_356 := TRUE;
   Ch3_DB2_358 := TRUE;
   Ch3_DB2_360 := TRUE;
   Ch3_DB2_362 := TRUE;
   Ch4_DB2_364 := TRUE;
   Ch4_DB2_366 := TRUE;
   Ch4_DB2_367 := TRUE;
   Ch4_DB2_370 := TRUE;
   Ch4_DB2_371 := TRUE;
   Ch4_DB2_374 := TRUE;
   Ch4_DB2_376 := TRUE;
   Ch4_DB2_378 := TRUE;
   Ch4_DB2_380 := TRUE;
   Ch5_DB2_382 := TRUE;
   Ch5_DB2_384 := TRUE;
   Ch5_DB2_385 := TRUE;
   Ch5_DB2_388 := TRUE;
   Ch5_DB2_389 := TRUE;
   Ch5_DB2_392 := TRUE;
   Ch5_DB2_394 := TRUE;
   Ch5_DB2_396 := TRUE;
   Ch5_DB2_398 := TRUE;
   Ch6_DB2_400 := TRUE;
   Ch6_DB2_402 := TRUE;
   Ch6_DB2_403 := TRUE;
   Ch6_DB2_406 := TRUE;
   Ch6_DB2_407 := TRUE;
   Ch6_DB2_410 := TRUE;
   Ch6_DB2_412 := TRUE;
   Ch6_DB2_414 := TRUE;
   Ch6_DB2_416 := TRUE;
   Ch7_DB2_418 := TRUE;
   Ch7_DB2_420 := TRUE;
   Ch7_DB2_421 := TRUE;
   Ch7_DB2_424 := TRUE;
   Ch7_DB2_425 := TRUE;
   Ch7_DB2_428 := TRUE;
   Ch7_DB2_430 := TRUE;
   Ch7_DB2_432 := TRUE;
   Ch7_DB2_434 := TRUE;
   Ch8_DB2_436 := TRUE;
   Ch8_DB2_438 := TRUE;
   Ch8_DB2_439 := TRUE;
   Ch8_DB2_442 := TRUE;
   Ch8_DB2_443 := TRUE;
   Ch8_DB2_446 := TRUE;
   Ch8_DB2_448 := TRUE;
   Ch8_DB2_450 := TRUE;
   Ch8_DB2_452 := TRUE;
   Ch9_DB2_454 := TRUE;
   Ch9_DB2_456 := TRUE;
   Ch9_DB2_457 := TRUE;
   Ch9_DB2_460 := TRUE;
   Ch9_DB2_461 := TRUE;
   Ch9_DB2_464 := TRUE;
   Ch9_DB2_466 := TRUE;
   Ch9_DB2_468 := TRUE;
   Ch9_DB2_470 := TRUE;
   Ch10_DB2_472 := TRUE;
   Ch10_DB2_474 := TRUE;
   Ch10_DB2_475 := TRUE;
   Ch10_DB2_478 := TRUE;
   Ch10_DB2_479 := TRUE;
   Ch10_DB2_482 := TRUE;
   Ch10_DB2_484 := TRUE;
   Ch10_DB2_486 := TRUE;
   Ch10_DB2_488 := TRUE;
   Ax1_DB2_490 := TRUE;
   Ax2_DB2_492 := TRUE;
   Ax3_DB2_494 := TRUE;
   Ax4_DB2_496 := TRUE;
   Ax5_DB2_498 := TRUE;
   Ax6_DB2_500 := TRUE;
   Ax7_DB2_502 := TRUE;
   Ax8_DB2_504 := TRUE;
   Ax9_DB2_506 := TRUE;
   Ax10_DB2_508 := TRUE;
   Ax11_DB2_510 := TRUE;
   Ax12_DB2_512 := TRUE;
   Ax13_DB2_514 := TRUE;
   Ax14_DB2_516 := TRUE;
   Ax15_DB2_518 := TRUE;
   Ax16_DB2_520 := TRUE;
   Ax17_DB2_522 := TRUE;
   Ax18_DB2_524 := TRUE;
   Ax19_DB2_526 := TRUE;
   Ax20_DB2_528 := TRUE;
   Ax21_DB2_530 := TRUE;
   Ax22_DB2_532 := TRUE;
   Ax23_DB2_534 := TRUE;
   Ax24_DB2_536 := TRUE;
   Ax25_DB2_538 := TRUE;
   Ax26_DB2_540 := TRUE;
   Ax27_DB2_542 := TRUE;
   Ax28_DB2_544 := TRUE;
   Ax29_DB2_546 := TRUE;
   Ax30_DB2_548 := TRUE;
   Ax31_DB2_550 := TRUE;
   Ax32_DB2_552 := TRUE;
   User0_DB2_554 := TRUE;
   User0_DB2_555 := TRUE;
   User0_DB2_556 := TRUE;
   User0_DB2_557 := TRUE;
   User1_DB2_562 := TRUE;
   User1_DB2_563 := TRUE;
   User1_DB2_564 := TRUE;
   User1_DB2_565 := TRUE;
   User2_DB2_570 := TRUE;
   User2_DB2_571 := TRUE;
   User2_DB2_572 := TRUE;
   User2_DB2_573 := TRUE;
   User3_DB2_578 := TRUE;
   User3_DB2_579 := TRUE;
   User3_DB2_580 := TRUE;
   User3_DB2_581 := TRUE;
   User4_DB2_586 := TRUE;
   User4_DB2_587 := TRUE;
   User4_DB2_588 := TRUE;
   User4_DB2_589 := TRUE;
   User5_DB2_594 := TRUE;
   User5_DB2_595 := TRUE;
   User5_DB2_596 := TRUE;
   User5_DB2_597 := TRUE;
   User6_DB2_602 := TRUE;
   User6_DB2_603 := TRUE;
   User6_DB2_604 := TRUE;
   User6_DB2_605 := TRUE;
   User7_DB2_610 := TRUE;
   User7_DB2_611 := TRUE;
   User7_DB2_612 := TRUE;
   User7_DB2_613 := TRUE;
   User8_DB2_618 := TRUE;
   User8_DB2_619 := TRUE;
   User8_DB2_620 := TRUE;
   User8_DB2_621 := TRUE;
   User9_DB2_626 := TRUE;
   User9_DB2_627 := TRUE;
   User9_DB2_628 := TRUE;
   User9_DB2_629 := TRUE;
   User10_DB2_634 := TRUE;
   User10_DB2_635 := TRUE;
   User10_DB2_636 := TRUE;
   User10_DB2_637 := TRUE;
   User11_DB2_642 := TRUE;
   User11_DB2_643 := TRUE;
   User11_DB2_644 := TRUE;
   User11_DB2_645 := TRUE;
   User12_DB2_650 := TRUE;
   User12_DB2_651 := TRUE;
   User12_DB2_652 := TRUE;
   User12_DB2_653 := TRUE;
   User13_DB2_658 := TRUE;
   User13_DB2_659 := TRUE;
   User13_DB2_660 := TRUE;
   User13_DB2_661 := TRUE;
   User14_DB2_666 := TRUE;
   User14_DB2_667 := TRUE;
   User14_DB2_668 := TRUE;
   User14_DB2_669 := TRUE;
   User15_DB2_674 := TRUE;
   User15_DB2_675 := TRUE;
   User15_DB2_676 := TRUE;
   User15_DB2_677 := TRUE;
   User16_DB2_682 := TRUE;
   User16_DB2_683 := TRUE;
   User16_DB2_684 := TRUE;
   User16_DB2_685 := TRUE;
   User17_DB2_690 := TRUE;
   User17_DB2_691 := TRUE;
   User17_DB2_692 := TRUE;
   User17_DB2_693 := TRUE;
   User18_DB2_698 := TRUE;
   User18_DB2_699 := TRUE;
   User18_DB2_700 := TRUE;
   User18_DB2_701 := TRUE;
   User19_DB2_706 := TRUE;
   User19_DB2_707 := TRUE;
   User19_DB2_708 := TRUE;
   User19_DB2_709 := TRUE;
   User20_DB2_714 := TRUE;
   User20_DB2_715 := TRUE;
   User20_DB2_716 := TRUE;
   User20_DB2_717 := TRUE;
   User21_DB2_722 := TRUE;
   User21_DB2_723 := TRUE;
   User21_DB2_724 := TRUE;
   User21_DB2_725 := TRUE;
   User22_DB2_730 := TRUE;
   User22_DB2_731 := TRUE;
   User22_DB2_732 := TRUE;
   User22_DB2_733 := TRUE;
   User23_DB2_738 := TRUE;
   User23_DB2_739 := TRUE;
   User23_DB2_740 := TRUE;
   User23_DB2_741 := TRUE;
   User24_DB2_746 := TRUE;
   User24_DB2_747 := TRUE;
   User24_DB2_748 := TRUE;
   User24_DB2_749 := TRUE;
   User25_DB2_754 := TRUE;
   User25_DB2_755 := TRUE;
   User25_DB2_756 := TRUE;
   User25_DB2_757 := TRUE;
   User26_DB2_762 := TRUE;
   User26_DB2_763 := TRUE;
   User26_DB2_764 := TRUE;
   User26_DB2_765 := TRUE;
   User27_DB2_770 := TRUE;
   User27_DB2_771 := TRUE;
   User27_DB2_772 := TRUE;
   User27_DB2_773 := TRUE;
   User28_DB2_778 := TRUE;
   User28_DB2_779 := TRUE;
   User28_DB2_780 := TRUE;
   User28_DB2_781 := TRUE;
   User29_DB2_786 := TRUE;
   User29_DB2_787 := TRUE;
   User29_DB2_788 := TRUE;
   User29_DB2_789 := TRUE;
   User30_DB2_794 := TRUE;
   User30_DB2_795 := TRUE;
   User30_DB2_796 := TRUE;
   User30_DB2_797 := TRUE;
   User31_DB2_802 := TRUE;
   User31_DB2_803 := TRUE;
   User31_DB2_804 := TRUE;
   User31_DB2_805 := TRUE;
END_DATA_BLOCK

DATA_BLOCK "gp_par"	// DB 7
TITLE = Parameters for Baseprogram
AUTHOR : NUMERIK
FAMILY : _800D
NAME : Basics
VERSION : 2.7
"RUN_UP"
BEGIN
END_DATA_BLOCK

DATA_BLOCK DB 8
AUTHOR : NUMERIK
FAMILY : _800D
NAME : Basics
VERSION : 2.7
  STRUCT
   Fc19_1 : ARRAY  [0 .. 3 ] OF BYTE ;
   Res0 : ARRAY  [0 .. 3 ] OF BYTE ;
   plData : ARRAY  [8 .. 43 ] OF BYTE ;
   TestAuto : BYTE ;
   FirstCycle : BYTE ;
   Res4 : WORD ;
   Res5 : BYTE ;
   IsFb15Correct : BYTE ;
   Res6 : ARRAY  [50 .. 61 ] OF BYTE ;
   Fc19_2 : ARRAY  [0 .. 3 ] OF BYTE ;
   Res8 : ARRAY  [66 .. 81 ] OF BYTE ;
   S7_error_id : WORD ;
   S7_error_param : WORD ;
   S7_error_adr : DWORD ;
   MinCycleTime : INT ;
   AdaptTime : INT ;
   ActCycleTime : INT ;
  END_STRUCT ;	
BEGIN
END_DATA_BLOCK

DATA_BLOCK DB 15
AUTHOR : NUMERIK
FAMILY : _800D
NAME : Bas_Com
VERSION : 2.7
  STRUCT
   fifoFull : BOOL ;
   readOffset : BYTE ;
   writeOffset : BYTE ;
   filler : BYTE ;
   Fifo : ARRAY  [1 .. 10 ] OF BYTE ;
   pduRefArr : ARRAY  [1 .. 12 ] OF //Little Endian Werte
   STRUCT
    diNo : WORD ;
    diPartLen : WORD ;
    PdiBeg : DWORD ;
   END_STRUCT ;
  END_STRUCT ;	
BEGIN
END_DATA_BLOCK

// DB 16: know-how protected block, not included

DATA_BLOCK "SPL"	// DB 18
TITLE = SPL dataarea
AUTHOR : NUMERIK
FAMILY : _800D
NAME : Basics
VERSION : 2.7
  STRUCT
   INSEP_VALID : ARRAY  [1 .. 8 ] OF BOOL ;	//used external SPL-Inputbytes(HW)
   OUTSEP_VALID : ARRAY  [1 .. 8 ] OF BOOL ;	//used external SPL-Outputbytes(HW)
   INSEP_ADDR : ARRAY  [1 .. 8 ] OF INT ;	//Addresses external SPL-Inputbytes(HW)
   OUTSEP_ADDR : ARRAY  [1 .. 8 ] OF INT ;	//Addresses external SPL-Outputbytes(HW)
   SPL_READY : BOOL ;	//setup finished
   STOP_MODE : BOOL ;	//0= Stop D, 1=Stop E
   SPL_DATA : STRUCT
    INSEP : ARRAY  [1 .. 64 ] OF BOOL ;
    OUTSEP : ARRAY  [1 .. 64 ] OF BOOL ;
    INSIP : ARRAY  [1 .. 64 ] OF BOOL ;
    OUTSIP : ARRAY  [1 .. 64 ] OF BOOL ;
    MARKERSIP : ARRAY  [1 .. 64 ] OF BOOL ;
   END_STRUCT ;
   SPL_DELTA : STRUCT 	//edge difference NCK - PLC for Diagnostic
    INSEP : ARRAY  [1 .. 64 ] OF BOOL ;
    OUTSEP : ARRAY  [1 .. 64 ] OF BOOL ;
    INSIP : ARRAY  [1 .. 64 ] OF BOOL ;
    OUTSIP : ARRAY  [1 .. 64 ] OF BOOL ;
    MARKERSIP : ARRAY  [1 .. 64 ] OF BOOL ;
   END_STRUCT ;
   CMDSI : BOOL ;	//multiplication of Timeout Value by Factor 10
   CMDSI_R1 : BOOL ;	//for future use
   CMDSI_R2 : BOOL ;	//for future use
   CMDSI_R3 : BOOL ;	//for future use
   CMDSI_R4 : BOOL ;	//for future use
   CMDSI_R5 : BOOL ;	//for future use
   CMDSI_R6 : BOOL ;	//for future use
   CMDSI_R7 : BOOL ;	//for future use
   STATUS_R0 : BOOL ;	//for future use
   STATUS_R1 : BOOL ;	//for future use
   STATUS_R2 : BOOL ;	//for future use
   STATUS_R3 : BOOL ;	//for future use
   STATUS_R4 : BOOL ;	//for future use
   COMM_TO : BOOL ;	//Communication Timeout
   STATUS_R6 : BOOL ;	//for future use
   STATUS_R7 : BOOL ;	//for future use
   STATSI : DINT ;	//Status: 0 - no error, 1 - 320 error number
   LEVELSI : DINT ;	//stacklevel SPL-KDV for Diagnostic
   PLCSIOUT : ARRAY  [1 .. 32 ] OF BOOL ;	//Single Channel Signals from NCK
   PLCSIIN : ARRAY  [1 .. 32 ] OF BOOL ;	//Single Channel Signals to NCK
   SPL_STATUS : ARRAY  [1 .. 16 ] OF BOOL ;	//SPL Status from NCK
   INSEP_PROFISAFE : ARRAY  [1 .. 8 ] OF BOOL ;	//external SPL-Inputbytes(HW) with PROFIsafe Slaves
   OUTSEP_PROFISAFE : ARRAY  [1 .. 8 ] OF BOOL ;	//external SPL-Outputbytes(HW) with PROFIsafe Slaves
   NoOfAxisPerBlock : ARRAY  [1 .. 8 ] OF BYTE ;	//Pointer and Tables for Teststop
   BlockPointer : ARRAY  [1 .. 8 ] OF BYTE ;
   AxisTable : ARRAY  [1 .. 31 ] OF BYTE ;
   FSDP : ARRAY  [1 .. 3 ] OF STRUCT
    ERR_REAC : INT ;	// IN: Error reaction
    ERROR : BOOL ;	// OUT: 1=Communication error
    SUBS_ON : BOOL ;	// OUT: 1=Receiver outputs fail-safe values
    DIAG : WORD ;	// OUT: Service information
    RETVAL14 : WORD ;	// OUT: Error code of SFC 14
    RETVAL15 : WORD ;	// OUT: Error code of SFC 15
   END_STRUCT ;
   FRDP : ARRAY  [1 .. 3 ] OF STRUCT
    SUBS : ARRAY  [0 .. 15 ] OF BOOL ;	// IN: Fail-safe value for receive data BOOL 00 ... BOOL 15
    ERR_REAC : INT ;	// IN: Error reaction
    ACK_REI : BOOL ;	// IN: 1=Acknowledgment for reintegration of send data following communication er
    RES1 : BOOL ;	//Reserved
    RES2 : BOOL ;	//Reserved
    RES3 : BOOL ;	//Reserved
    RES4 : BOOL ;	//Reserved
    RES5 : BOOL ;	//Reserved
    RES6 : BOOL ;	//Reserved
    RES7 : BOOL ;	//Reserved
    ERROR : BOOL ;	// OUT: 1=Communication error
    SUBS_ON : BOOL ;	// OUT: 1=Fail-safe values are output
    ACK_REQ : BOOL ;	// OUT: 1=Acknowledgment for reintegration of send data required
    SENDMODE : BOOL ;	// OUT: 1=F_CPU with F_SENDDP in deactivated safety mode
    DIAG : WORD ;	// OUT: Service information
    RETVAL14 : WORD ;	// OUT: Error code of SFC 14
    RETVAL15 : WORD ;	// OUT: Error code of SFC 15
   END_STRUCT ;
   SPL_USER_DATA : ARRAY  [0 .. 3 ] OF DWORD ;
  END_STRUCT ;	
BEGIN
END_DATA_BLOCK

DATA_BLOCK "CtrlE"	// DB 1000
TITLE = Datainterface Ctrl-Energy
AUTHOR : NUMERIK
FAMILY : _800D
NAME : CTRL_E
VERSION : 2.7
  STRUCT
   Profile : ARRAY  [1 .. 8 ] OF STRUCT
    ESaveOn : BOOL ;	// Activate energy-saving profile immediately
    ReloadT2 : BOOL ;	// Reload Prewarning time (T2)
    res0_2 : BOOL ;
    res0_3 : BOOL ;
    res0_4 : BOOL ;
    res0_5 : BOOL ;
    res0_6 : BOOL ;
    res0_7 : BOOL ;
    HmiESaveOn : BOOL ;	// HMI->PLC: Activate energy-saving profile immediately
    res1_1 : BOOL ;
    res1_2 : BOOL ;
    res1_3 : BOOL ;
    res1_4 : BOOL ;
    res1_5 : BOOL ;
    res1_6 : BOOL ;
    res1_7 : BOOL ;
    MasterCompSig : BOOL ;	// Master computer signal
    PlcUserSig : BOOL ;	// PLC user signal
    res2_2 : BOOL ;
    res2_3 : BOOL ;
    res2_4 : BOOL ;
    res2_5 : BOOL ;
    res2_6 : BOOL ;
    res2_7 : BOOL ;
    res3 : BYTE ;
    ESaveIsOn : BOOL ;	// Energy-saving state active
    T1Expired : BOOL ;	// Activation time T1 expired
    res4_2 : BOOL ;
    res4_3 : BOOL ;
    res4_4 : BOOL ;
    res4_5 : BOOL ;
    res4_6 : BOOL ;
    res4_7 : BOOL ;
    res5 : BYTE ;
    ActValT1 : INT ;	// T1 current value
    ActValT2 : INT ;	// T2 current value
    ESaveValid : BOOL ;	// HMI->PLC: Energy-saving profile valid
    ESaveOff : BOOL ;	// HMI->PLC: Deactivate energy-saving profileblock energy-saving profile
    res10_2 : BOOL ;
    res10_3 : BOOL ;
    res10_4 : BOOL ;
    res10_5 : BOOL ;
    res10_6 : BOOL ;
    res10_7 : BOOL ;
    CondOpPanel : BOOL ;	// HMI->PLC: Operator panel
    CondDataTransfer : BOOL ;	// HMI->PLC: Data transfer
    CondWindowChange : BOOL ;	// HMI->PLC: Window change
    res11_3 : BOOL ;
    res11_4 : BOOL ;
    res11_5 : BOOL ;
    res11_6 : BOOL ;
    res11_7 : BOOL ;
    CondMCP : BOOL ;	// HMI->PLC: Machine control panel
    res12_1 : BOOL ;
    res12_2 : BOOL ;
    res12_3 : BOOL ;
    res12_4 : BOOL ;
    res12_5 : BOOL ;
    res12_6 : BOOL ;
    res12_7 : BOOL ;
    CondNcChan1 : BOOL ;	// HMI->PLC: NC channel 1 in reset
    CondNcChan2 : BOOL ;	// HMI->PLC: NC channel 2 in reset
    CondNcChan3 : BOOL ;	// HMI->PLC: NC channel 3 in reset
    CondNcChan4 : BOOL ;	// HMI->PLC: NC channel 4 in reset
    CondNcChan5 : BOOL ;	// HMI->PLC: NC channel 5 in reset
    CondNcChan6 : BOOL ;	// HMI->PLC: NC channel 6 in reset
    CondNcChan7 : BOOL ;	// HMI->PLC: NC channel 7 in reset
    CondNcChan8 : BOOL ;	// HMI->PLC: NC channel 8 in reset
    CondNcChan9 : BOOL ;	// HMI->PLC: NC channel 9 in reset
    CondNcChan10 : BOOL ;	// HMI->PLC: NC channel 10 in reset
    res14_2 : BOOL ;
    res14_3 : BOOL ;
    res14_4 : BOOL ;
    res14_5 : BOOL ;
    res14_6 : BOOL ;
    res14_7 : BOOL ;
    CondMasterCompSig : BOOL ;	// HMI->PLC: Master computer signal
    CondPlcUserSig : BOOL ;	// HMI->PLC: PLC user signal
    res15_2 : BOOL ;
    res15_3 : BOOL ;
    res15_4 : BOOL ;
    res15_5 : BOOL ;
    res15_6 : BOOL ;
    res15_7 : BOOL ;
    PresetT1 : INT ;	// HMI->PLC: Activation time T1
    PresetT2 : INT ;	// HMI->PLC: Prewarning time T2
   END_STRUCT ;
  END_STRUCT ;	
BEGIN
   Profile[1].ESaveValid := TRUE;
   Profile[1].ESaveOff := TRUE;
   Profile[1].CondNcChan1 := TRUE;
   Profile[1].CondNcChan2 := TRUE;
   Profile[1].CondNcChan3 := TRUE;
   Profile[1].CondNcChan4 := TRUE;
   Profile[1].CondNcChan5 := TRUE;
   Profile[1].CondNcChan6 := TRUE;
   Profile[1].CondNcChan7 := TRUE;
   Profile[1].CondNcChan8 := TRUE;
   Profile[1].CondNcChan9 := TRUE;
   Profile[1].CondNcChan10 := TRUE;
   Profile[1].CondPlcUserSig := TRUE;
   Profile[1].PresetT1 := 60;
   Profile[1].PresetT2 := 120;
   Profile[2].ESaveValid := TRUE;
   Profile[2].ESaveOff := TRUE;
   Profile[2].CondMCP := TRUE;
   Profile[2].CondNcChan1 := TRUE;
   Profile[2].CondNcChan2 := TRUE;
   Profile[2].CondNcChan3 := TRUE;
   Profile[2].CondNcChan4 := TRUE;
   Profile[2].CondNcChan5 := TRUE;
   Profile[2].CondNcChan6 := TRUE;
   Profile[2].CondNcChan7 := TRUE;
   Profile[2].CondNcChan8 := TRUE;
   Profile[2].CondNcChan9 := TRUE;
   Profile[2].CondNcChan10 := TRUE;
   Profile[2].CondPlcUserSig := TRUE;
   Profile[2].PresetT1 := 120;
   Profile[2].PresetT2 := 300;
   Profile[3].ESaveValid := TRUE;
   Profile[3].ESaveOff := TRUE;
   Profile[3].CondOpPanel := TRUE;
   Profile[3].CondDataTransfer := TRUE;
   Profile[3].CondWindowChange := TRUE;
   Profile[3].CondMCP := TRUE;
   Profile[3].CondNcChan1 := TRUE;
   Profile[3].CondNcChan2 := TRUE;
   Profile[3].CondNcChan3 := TRUE;
   Profile[3].CondNcChan4 := TRUE;
   Profile[3].CondNcChan5 := TRUE;
   Profile[3].CondNcChan6 := TRUE;
   Profile[3].CondNcChan7 := TRUE;
   Profile[3].CondNcChan8 := TRUE;
   Profile[3].CondNcChan9 := TRUE;
   Profile[3].CondNcChan10 := TRUE;
   Profile[3].CondPlcUserSig := TRUE;
   Profile[3].PresetT1 := 600;
END_DATA_BLOCK

DATA_BLOCK "SentronPac"	// DB 1001
TITLE = Datainterface SentronPac
AUTHOR : NUMERIK
FAMILY : _800D
NAME : SENTRONP
VERSION : 2.7
  STRUCT
   ManualVal : BOOL ;	// Display of manual value
   SentronPacMach : BOOL ;	// Sentron PAC represented machine
   FeedInEnergyReadSP : BOOL ;	// Feed in energy read from Sentron PAC
   FeedBackEnergyReadSP : BOOL ;	// Feed back energy read from Sentron PAC
   res1 : BYTE ;
   MeasAct : BOOL ;	// Active measurement
   res3 : BYTE ;
   ManualValue : REAL ;	// Manual value
   ActivePowerItem : REAL ;	// Active power item
   ActiveEnergyItem : REAL ;	// Active energy item
   ReactiveEnergyItem : REAL ;	// Reactive energy item
  END_STRUCT ;	
BEGIN
END_DATA_BLOCK

ORGANIZATION_BLOCK OB 1
VERSION : 1.0
VAR_TEMP
  OB1_EV_CLASS : BYTE ;
  OB1_SCAN_1 : BYTE ;
  OB1_PRIORITY : BYTE ;
  OB1_OB_NUMBR : BYTE ;
  OB1_RESERVED_1 : BYTE ;
  OB1_RESERVED_2 : BYTE ;
  OB1_PREV_CYCLE : INT ;
  OB1_MIN_CYCLE : INT ;
  OB1_MAX_CYCLE : INT ;
  OB1_DATE_TIME : DATE_AND_TIME ;
END_VAR
BEGIN
NETWORK
TITLE =
      CALL  "GP_HP";
//Insert User program from here
END_ORGANIZATION_BLOCK

ORGANIZATION_BLOCK OB 40
VERSION : 1.0
VAR_TEMP
  OB40_EV_CLASS : BYTE ;
  OB40_STRT_INF : BYTE ;
  OB40_PRIORITY : BYTE ;
  OB40_OB_NUMBR : BYTE ;
  OB40_RESERVED_1 : BYTE ;
  OB40_MDL_ID : BYTE ;
  OB40_MDL_ADDR : INT ;
  OB40_POINT_ADDR : DWORD ;
  OB40_DATE_TIME : DATE_AND_TIME ;	//data for the Basic program
  GP_IRFromNCK : BOOL ;	//Interrupt from NCK
  GP_TM : BOOL ;	//Toolmanagment
  GP_InPosition : ARRAY  [1 .. 31 ] OF BOOL ;	//InPos Signal from FC15,16,18
  GP_AuxFunction : ARRAY  [1 .. 10 ] OF BOOL ;	//auxiliary functions
  GP_FMBlock : ARRAY  [1 .. 10 ] OF BOOL ;	//not used
//Insert User-data from here
END_VAR
BEGIN
NETWORK
TITLE =
      CALL  "GP_PRAL";
//Insert User program from here
END_ORGANIZATION_BLOCK

ORGANIZATION_BLOCK OB 82
TITLE = "I/O Point Fault"
VERSION : 1.0
VAR_TEMP
  OB82_EV_CLASS : BYTE ;	//16#39, Event class 3, Entering event state, Internal fault event
  OB82_FLT_ID : BYTE ;	//16#XX, Fault identifcation code
  OB82_PRIORITY : BYTE ;	//Priority of OB Execution
  OB82_OB_NUMBR : BYTE ;	//82 (Organization block 82, OB82)
  OB82_RESERVED_1 : BYTE ;	//Reserved for system
  OB82_IO_FLAG : BYTE ;	//Input (01010100), Output (01010101)
  OB82_MDL_ADDR : WORD ;	//Base address of module with fault
  OB82_MDL_DEFECT : BOOL ;	//Module defective
  OB82_INT_FAULT : BOOL ;	//Internal fault
  OB82_EXT_FAULT : BOOL ;	//External fault
  OB82_PNT_INFO : BOOL ;	//Point information
  OB82_EXT_VOLTAGE : BOOL ;	//External voltage low
  OB82_FLD_CONNCTR : BOOL ;	//Field wiring connector missing
  OB82_NO_CONFIG : BOOL ;	//Module has no configuration data
  OB82_CONFIG_ERR : BOOL ;	//Module has configuration error
  OB82_MDL_TYPE : BYTE ;	//Type of module
  OB82_SUB_MDL_ERR : BOOL ;	//Sub-Module is missing or has error
  OB82_COMM_FAULT : BOOL ;	//Communication fault
  OB82_MDL_STOP : BOOL ;	//Module is stopped
  OB82_WTCH_DOG_FLT : BOOL ;	//Watch dog timer stopped module
  OB82_INT_PS_FLT : BOOL ;	//Internal power supply fault
  OB82_PRIM_BATT_FLT : BOOL ;	//Primary battery is in fault
  OB82_BCKUP_BATT_FLT : BOOL ;	//Backup battery is in fault
  OB82_RESERVED_2 : BOOL ;	//Reserved for system
  OB82_RACK_FLT : BOOL ;	//Rack fault, only for bus interface module
  OB82_PROC_FLT : BOOL ;	//Processor fault
  OB82_EPROM_FLT : BOOL ;	//EPROM fault
  OB82_RAM_FLT : BOOL ;	//RAM fault
  OB82_ADU_FLT : BOOL ;	//ADU fault
  OB82_FUSE_FLT : BOOL ;	//Fuse fault
  OB82_HW_INTR_FLT : BOOL ;	//Hardware interupt input in fault
  OB82_RESERVED_3 : BOOL ;	//Reserved for system
  OB82_DATE_TIME : DATE_AND_TIME ;	//Date and time OB82 started
END_VAR
BEGIN
NETWORK
TITLE = Detailed Diagnosis in OB82 (interrupt)
      CALL  "GP_DIAG" (
           $1                       := TRUE);
END_ORGANIZATION_BLOCK

ORGANIZATION_BLOCK OB 86
TITLE = "Loss Of Rack Fault"
VERSION : 1.0
VAR_TEMP
  OB86_EV_CLASS : BYTE ;	//16#38/39 Event class 3
  OB86_FLT_ID : BYTE ;	//16#C1/C4/C5, Fault identifcation code
  OB86_PRIORITY : BYTE ;	//Priority of OB Execution
  OB86_OB_NUMBR : BYTE ;	//86 (Organization block 86, OB86)
  OB86_RESERVED_1 : BYTE ;	//Reserved for system
  OB86_RESERVED_2 : BYTE ;	//Reserved for system
  OB86_MDL_ADDR : WORD ;	//Base address of IM module in rack with fault
  OB86_RACKS_FLTD : ARRAY  [0 .. 31 ] OF BOOL ;	//Racks in fault
  OB86_DATE_TIME : DATE_AND_TIME ;	//Date and time OB86 started
END_VAR
BEGIN
NETWORK
TITLE = Detailed Diagnosis in OB86 (interrupt)
      CALL  "GP_DIAG" (
           $1                       := TRUE);
END_ORGANIZATION_BLOCK

ORGANIZATION_BLOCK OB 100
VERSION : 1.0
VAR_TEMP
  OB100_EV_CLASS : BYTE ;
  OB100_STRTUP : BYTE ;
  OB100_PRIORITY : BYTE ;
  OB100_OB_NUMBR : BYTE ;
  OB100_RESERVED_1 : BYTE ;
  OB100_RESERVED_2 : BYTE ;
  OB100_STOP : WORD ;
  OB100_RESERVED_3 : WORD ;
  OB100_RESERVED_4 : WORD ;
  OB100_DATE_TIME : DATE_AND_TIME ;
END_VAR
BEGIN
NETWORK
TITLE =
      CALL  "RUN_UP" , "gp_par" (
           DIW 0                    := 1,
           DIW 2                    := 0,
           DID 4                    := P#I 0.0,
           DIW 8                    := 0,
           DID 10                   := P#Q 0.0,
           DIW 14                   := 0,
           DID 16                   := P#Q 8.0,
           DIW 20                   := 0,
           DID 22                   := P#Q 12.0,
           DIW 26                   := 6);
//Insert User program from here
END_ORGANIZATION_BLOCK
